	//Aktivera Utsignal Y1
	FB_MBReadCoils_Y1(
		sIPAddr:= sIpAddr, 
		nTCPPort:= INT_TO_UINT(nTCPPort), 
		nUnitID:= INT_TO_BYTE(nUnitID), 
		nQuantity:=1, 
		nMBAddr:= 0, 
		cbLength:= SIZEOF(bY1EnableRead), 
		pDestAddr:= ADR(bY1EnableRead), 
		bExecute:= bSekvensFlagga, 
		tTimeout:= T#3S, 
		bBusy=> , 
		bError=> , 
		nErrId=> , 
		cbRead=> );
				
		IF bY1Enable <> bY1EnableRead AND bSekvensFlagga THEN
			FB_MBWriteCoils_Y1.bExecute := TRUE;
		ELSE
			FB_MBWriteCoils_Y1.bExecute := FALSE;
		END_IF
		
	FB_MBWriteCoils_Y1(
		sIPAddr:= sIpAddr, 
		nTCPPort:= INT_TO_UINT(nTCPPort), 
		nUnitID:= INT_TO_BYTE(nUnitID), 
		nQuantity:= 1, 
		nMBAddr:= 0, 
		cbLength:= SIZEOF(bY1Enable), 
		pSrcAddr:= ADR(bY1Enable), 
		bExecute:= , 
		tTimeout:= , 
		bBusy=> , 
		bError=> , 
		nErrId=> );	
		
	//Aktivera Utsignal Y2
	FB_MBReadCoils_Y2(
		sIPAddr:= sIpAddr, 
		nTCPPort:= INT_TO_UINT(nTCPPort), 
		nUnitID:= INT_TO_BYTE(nUnitID), 
		nQuantity:=1, 
		nMBAddr:= 1, 
		cbLength:= SIZEOF(bY2EnableRead), 
		pDestAddr:= ADR(bY2EnableRead), 
		bExecute:= bSekvensFlagga, 
		tTimeout:= T#3S, 
		bBusy=> , 
		bError=> , 
		nErrId=> , 
		cbRead=> );
				
		IF bY2Enable <> bY2EnableRead AND bSekvensFlagga THEN
			FB_MBWriteCoils_Y2.bExecute := TRUE;
		ELSE
			FB_MBWriteCoils_Y2.bExecute := FALSE;
		END_IF
		
	FB_MBWriteCoils_Y2(
		sIPAddr:= sIpAddr, 
		nTCPPort:= INT_TO_UINT(nTCPPort), 
		nUnitID:= INT_TO_BYTE(nUnitID), 
		nQuantity:= 1, 
		nMBAddr:= 1, 
		cbLength:= SIZEOF(bY2Enable), 
		pSrcAddr:= ADR(bY2Enable), 
		bExecute:= , 
		tTimeout:= , 
		bBusy=> , 
		bError=> , 
		nErrId=> );		
		
	//Aktivera Utsignal Y3
	FB_MBReadCoils_Y3(
		sIPAddr:= sIpAddr, 
		nTCPPort:= INT_TO_UINT(nTCPPort), 
		nUnitID:= INT_TO_BYTE(nUnitID), 
		nQuantity:=1, 
		nMBAddr:= 2, 
		cbLength:= SIZEOF(bY3EnableRead), 
		pDestAddr:= ADR(bY3EnableRead), 
		bExecute:= bSekvensFlagga, 
		tTimeout:= T#3S, 
		bBusy=> , 
		bError=> , 
		nErrId=> , 
		cbRead=> );
				
		IF bY3Enable <> bY3EnableRead AND bSekvensFlagga THEN
			FB_MBWriteCoils_Y3.bExecute := TRUE;
		ELSE
			FB_MBWriteCoils_Y3.bExecute := FALSE;
		END_IF
		
	FB_MBWriteCoils_Y3(
		sIPAddr:= sIpAddr, 
		nTCPPort:= INT_TO_UINT(nTCPPort), 
		nUnitID:= INT_TO_BYTE(nUnitID), 
		nQuantity:= 1, 
		nMBAddr:= 2, 
		cbLength:= SIZEOF(bY3Enable), 
		pSrcAddr:= ADR(bY3Enable), 
		bExecute:= , 
		tTimeout:= , 
		bBusy=> , 
		bError=> , 
		nErrId=> );		
		
	//Aktivera Utsignal Y4
	FB_MBReadCoils_Y4(
		sIPAddr:= sIpAddr, 
		nTCPPort:= INT_TO_UINT(nTCPPort), 
		nUnitID:= INT_TO_BYTE(nUnitID), 
		nQuantity:=1, 
		nMBAddr:= 3, 
		cbLength:= SIZEOF(bY4EnableRead), 
		pDestAddr:= ADR(bY4EnableRead), 
		bExecute:= bSekvensFlagga, 
		tTimeout:= T#3S, 
		bBusy=> , 
		bError=> , 
		nErrId=> , 
		cbRead=> );
				
		IF bY4Enable <> bY4EnableRead AND bSekvensFlagga THEN
			FB_MBWriteCoils_Y4.bExecute := TRUE;
		ELSE
			FB_MBWriteCoils_Y4.bExecute := FALSE;
		END_IF
		
	FB_MBWriteCoils_Y4(
		sIPAddr:= sIpAddr, 
		nTCPPort:= INT_TO_UINT(nTCPPort), 
		nUnitID:= INT_TO_BYTE(nUnitID), 
		nQuantity:= 1, 
		nMBAddr:= 3, 
		cbLength:= SIZEOF(bY4Enable), 
		pSrcAddr:= ADR(bY4Enable), 
		bExecute:= , 
		tTimeout:= , 
		bBusy=> , 
		bError=> , 
		nErrId=> );		

//Holding register

//Börvärde Y1
wTemp := OaksLibrary.fRealToWord(rReal:= rY1Setpoint, uiFaktor:= 10);
//rtemp := rY1Setpoint * 10;
//iTemp := LIMIT(0,REAL_TO_UINT(rtemp),1000);
		
//Skriv börvärde
fbReadWriteHoldingReg_Y1(
	sIPAddr:= sIpAddr, 
	nTCPPort:= INT_TO_UINT(nTCPPort), 
	nUnitID:= INT_TO_BYTE(nUnitID), 
	mBusAdr:= 0, 
	bEnable:= bSekvensFlagga AND bY1Enable, 
	iWrite:= wTemp, 
	iRead=> , 
	bError=> );

//Börvärde Y2
wTemp := OaksLibrary.fRealToWord(rReal:= rY2Setpoint, uiFaktor:= 10);
//rtemp := rY2Setpoint * 10;
//iTemp := LIMIT(0,REAL_TO_UINT(rtemp),1000);
		
//Skriv börvärde Setpoint
fbReadWriteHoldingReg_Y2(
	sIPAddr:= sIpAddr, 
	nTCPPort:= INT_TO_UINT(nTCPPort), 
	nUnitID:= INT_TO_BYTE(nUnitID), 
	mBusAdr:= 1, 
	bEnable:= bSekvensFlagga AND bY2Enable, 
	iWrite:= wTemp, 
	iRead=> , 
	bError=> );	

//Börvärde Y3
wTemp := OaksLibrary.fRealToWord(rReal:= rY3Setpoint, uiFaktor:= 10);	
//rtemp := rY3Setpoint * 10;
//iTemp := LIMIT(0,REAL_TO_UINT(rtemp),1000);
		
//Skriv börvärde Setpoint
fbReadWriteHoldingReg_Y3(
	sIPAddr:= sIpAddr, 
	nTCPPort:= INT_TO_UINT(nTCPPort), 
	nUnitID:= INT_TO_BYTE(nUnitID), 
	mBusAdr:= 2, 
	bEnable:= bSekvensFlagga AND bY3Enable, 
	iWrite:= wTemp, 
	iRead=> , 
	bError=> );	
	
//Börvärde Y4
wTemp := OaksLibrary.fRealToWord(rReal:= rY4Setpoint, uiFaktor:= 10);	
//rtemp := rY4Setpoint * 10;
//iTemp := LIMIT(0,REAL_TO_UINT(rtemp),1000);
		
//Skriv börvärde Setpoint
fbReadWriteHoldingReg_Y4(
	sIPAddr:= sIpAddr, 
	nTCPPort:= INT_TO_UINT(nTCPPort), 
	nUnitID:= INT_TO_BYTE(nUnitID), 
	mBusAdr:= 3, 
	bEnable:= bSekvensFlagga AND bY4Enable, 
	iWrite:= wTemp, 
	iRead=> , 
	bError=> );	
	
//Communication error
	fbKommTof(IN:=FB_MBReadRegs_InputRegs1.bError OR FB_MBReadCoils_Y1.bError OR FB_MBReadCoils_Y2.bError OR FB_MBReadCoils_Y3.bError OR FB_MBReadCoils_Y4.bError OR fbReadWriteHoldingReg_Y1.bError OR fbReadWriteHoldingReg_Y2.bError OR fbReadWriteHoldingReg_Y3.bError OR fbReadWriteHoldingReg_Y4.bError, PT:=T#20S , Q=> , ET=> );
	
	fbAlarm_1(bInput:= fbKommTof.Q, tAlarmDelay:= T#20M, bAutoReset:= TRUE, bAlarmOutput=> FAULT);
		
//Write busy	
	oaksgvl.aBModbusBusyFlagga[iModbusLoop,nUnitID] := FB_MBReadRegs_InputRegs1.bBusy OR FB_MBReadCoils_Y1.bBusy OR FB_MBReadCoils_Y2.bBusy OR FB_MBReadCoils_Y3.bBusy OR FB_MBReadCoils_Y4.bBusy OR fbReadWriteHoldingReg_Y1.bBusy OR fbReadWriteHoldingReg_Y2.bBusy OR fbReadWriteHoldingReg_Y3.bBusy OR fbReadWriteHoldingReg_Y4.bBusy;

END_FUNCTION_BLOCK

// oaksModbusLibrary/Produal/Regulatorer/fbProdualHdhmCo2PirOverride
FUNCTION_BLOCK fbProdualHdhmCo2PirOverride EXTENDS fbProdualHdhmCo2Override
VAR_INPUT 
END_VAR
VAR_OUTPUT
	V AT %M*: BOOL; //Närvaroindikering (fördröjt till och frånslag)~wp:[trendoptions]i:300
	PV4 AT %M*: BOOL; //Närvarogivare (Rå-värde)~wp:[trendoptions]i:300	
END_VAR
VAR
	fbReadPir : FB_MBReadInputs;
	
	fbWriteStartDelay : fbReadWriteHoldingRegReal;
	fbWriteStopDelay : fbReadWriteHoldingRegReal;
	bReadPir : BYTE; // 10002 PIR sensor state (immediate) - 10003 PIR sensor state (control)
END_VAR

VAR_INPUT PERSISTENT
	SP7 AT %M*: REAL; //Fördröjning aktivering närvaroindikering (0-1-2)~wp:[format]0
	SP8 AT %M*: REAL; //Fördröjning inaktivering närvaroindikering (0-1-2-3-4-5)~wp:[format]0
END_VAR

SUPER^();

	//Read Status
	fbReadPir(
	sIPAddr:= sIpAddr, 
	nTCPPort:= INT_TO_UINT(nTCPPort), 
	nUnitID:= INT_TO_BYTE(nUnitID), 
	nQuantity:= 2, 
	nMBAddr:= 1, 
	cbLength:= SIZEOF(bReadPir), 
	pDestAddr:= ADR(bReadPir), 
	bExecute:= bSekvensFlagga, 
	tTimeout:=T#20S , 
	bBusy=> , 
	bError=> , 
	nErrId=> , 
	cbRead=> );
	
	PV4 :=  bReadPir.0;
	V := bReadPir.1;

	//Start-/Stoppfördröjning
	
	fbWriteStartDelay(
	sIPAddr:= sIpAddr, 
	nTCPPort:= INT_TO_UINT(nTCPPort), 
	nUnitID:= INT_TO_BYTE(nUnitID), 
	mBusAdr:=34 , 
	bEnable:=bSekvensFlagga , 
	tTimeout:= T#3S, 
	rReal:= SP7, 
	uiFaktor:= 1, 
	bError=> , 
	bBusy=> , 
	bSuccess=> );
		
	fbWriteStopDelay(
	sIPAddr:= sIpAddr, 
	nTCPPort:= INT_TO_UINT(nTCPPort), 
	nUnitID:= INT_TO_BYTE(nUnitID), 
	mBusAdr:=35 , 
	bEnable:=bSekvensFlagga , 
	tTimeout:= T#3S, 
	rReal:= SP8, 
	uiFaktor:= 1, 
	bError=> , 
	bBusy=> , 
	bSuccess=> );

END_FUNCTION_BLOCK

// oaksModbusLibrary/Regin/Givare/fbCthrc
FUNCTION_BLOCK fbCthrc
VAR_INPUT
	sIPAddr : STRING := ''; 
	nTCPPort : UINT;
	nUnitID : UINT;
	iModbusLoop : INT :=1; //Modbusslinga
	tKommfelsLarm : TIME := T#20M;
END_VAR
VAR_OUTPUT
	PV AT %M* : REAL;//Rumstemperatur~wp:[unit]°C[format]0.0[trendoptions]i:300
	PV1 AT %M* : REAL;//Koldioxidhalt~wp:[unit]ppm[format]0[trendoptions]i:300
	PV2 AT %M* : REAL;//Fukthalt~wp:[unit]rH%[format]0[trendoptions]i:300
	PV8 AT %M* : STRING;//Modbus konfiguering~wp:
	FAULT AT %M* : BOOL;//Kommunikationsfel~wp:
END_VAR
VAR
	sIP: STRING(255);
	sPort: STRING(255);
	sModbusID: STRING(255);
	sModbusLoop: STRING(255);
	sTemp : STRING(255);

	rTemp : REAL;
	fbKommTof : tof; 
	fbKommTon : ton;
	fbTempCo2Humidity: FB_MBReadRegs;
	wTempCo2Humidity : ARRAY[0..2] OF WORD; 
	bSekvensFlagga : BOOL;
END_VAR

//Modbus konfiguering
	sIP := CONCAT (SIPAddr, '');
	sPort := CONCAT ('<br>Port: ', UINT_TO_STRING(nTCPPort)); 								
	sModbusID := CONCAT('<br>ID: ', UINT_TO_STRING(nUnitID));
	sModbusLoop := CONCAT('<br>Loop: ', INT_TO_STRING(iModbusLoop));	

	sTemp := sIP;
	sTemp := CONCAT(sTemp, sPort);
	sTemp := CONCAT(sTemp, sModbusID);
	sTemp := CONCAT(sTemp, sModbusLoop);
	
	PV8 := sTemp;

//Sekvens	
	bSekvensFlagga := oaksGVL.aBModbusSekvens[iModbusLoop] = UINT_TO_INT(nUnitID);	
	
fbTempCo2Humidity(
	sIPAddr:= sIpAddr, 
	nTCPPort:= INT_TO_UINT(nTCPPort), 
	nUnitID:= INT_TO_BYTE(nUnitID), 
	nQuantity:=3 , 
	nMBAddr:=3999 , 
	cbLength:= SIZEOF(wTempCo2Humidity), 
	pDestAddr:= ADR(wTempCo2Humidity), 
	bExecute:= bSekvensFlagga, 
	tTimeout:= T#4.5S, 
	bBusy=> , 
	bError=> , 
	nErrId=> , 
	cbRead=> );
	
	fbKommTof(IN:=fbTempCo2Humidity.bError , PT:=T#20S , Q=> , ET=> );
	fbKommTon(IN:=fbKommTof.Q , PT:=tKommfelsLarm , Q=> , ET=> );
	FAULT :=fbKommTon.Q;
	
	rTemp := wTempCo2Humidity[0];
	PV2 := rTemp / 10 ; 
	rTemp := wTempCo2Humidity[1];
	PV := rTemp / 10; 
	PV1 := wTempCo2Humidity[2];

	//Write busy	
	oaksgvl.aBModbusBusyFlagga[iModbusLoop,nUnitID] := fbTempCo2Humidity.bBusy;

END_FUNCTION_BLOCK

// oaksModbusLibrary/Regin/Givare/fbCtrc
FUNCTION_BLOCK fbCtrc
VAR_INPUT
	sIPAddr : STRING := ''; 
	nTCPPort : UINT;
	nUnitID : UINT;
	iModbusLoop : INT :=1; //Modbusslinga
	tKommfelsLarm : TIME := T#20M;
END_VAR
VAR_OUTPUT
	PV AT %M* : REAL;//Rumstemperatur~wp:[unit]°C[format]0.0[trendoptions]i:300
	PV1 AT %M* : REAL;//Koldioxidhalt~wp:[unit]ppm[trendoptions]i:300
	PV8 AT %M* : STRING;//Modbus konfiguering~wp:
	FAULT AT %M* : BOOL;//Kommunikationsfel~wp:


END_VAR
VAR
	sIP: STRING(255);
	sPort: STRING(255);
	sModbusID: STRING(255);
	sModbusLoop: STRING(255);
	sTemp : STRING(255);

	rTemp : REAL;
	fbKommTof : tof; 
	fbKommTon : ton;
	fbTempCo2Humidity: FB_MBReadRegs;
	wTempCo2Humidity : ARRAY[0..1] OF	WORD; 
	bSekvensFlagga : BOOL;
END_VAR

//Modbus konfiguering
	sIP := CONCAT (SIPAddr, '');
	sPort := CONCAT ('<br>Port: ', UINT_TO_STRING(nTCPPort)); 								
	sModbusID := CONCAT('<br>ID: ', UINT_TO_STRING(nUnitID));
	sModbusLoop := CONCAT('<br>Loop: ', INT_TO_STRING(iModbusLoop));	

	sTemp := sIP;
	sTemp := CONCAT(sTemp, sPort);
	sTemp := CONCAT(sTemp, sModbusID);
	sTemp := CONCAT(sTemp, sModbusLoop);
	
	PV8 := sTemp;

//Sekvens	
	bSekvensFlagga := oaksGVL.aBModbusSekvens[iModbusLoop] = UINT_TO_INT(nUnitID);	
	
fbTempCo2Humidity(
	sIPAddr:= sIpAddr, 
	nTCPPort:= INT_TO_UINT(nTCPPort), 
	nUnitID:= INT_TO_BYTE(nUnitID), 
	nQuantity:=2 , 
	nMBAddr:=4000 , 
	cbLength:= SIZEOF(wTempCo2Humidity), 
	pDestAddr:= ADR(wTempCo2Humidity), 
	bExecute:= bSekvensFlagga, 
	tTimeout:= T#3S, 
	bBusy=> , 
	bError=> , 
	nErrId=> , 
	cbRead=> );
	
	fbKommTof(IN:=fbTempCo2Humidity.bError , PT:=T#20S , Q=> , ET=> );
	fbKommTon(IN:=fbKommTof.Q , PT:=tKommfelsLarm , Q=> , ET=> );
	FAULT :=fbKommTon.Q;
	
	
	rTemp := wTempCo2Humidity[0];
	PV := rTemp / 10; 
	PV1 := wTempCo2Humidity[1];

	//Write busy	
	oaksgvl.aBModbusBusyFlagga[iModbusLoop,nUnitID] := fbTempCo2Humidity.bBusy;

END_FUNCTION_BLOCK

// oaksModbusLibrary/Regin/Regio midi/fbReginRCC
//OAKS AB
//2020-04-28
//Funktionsblock för modbus-TCP, Regin RCC-C3DOCS rumsreglator med kyla/värme/spjäll. Inbyggda larm för hög/låg rumstemperatur och hög CO2-halt.
FUNCTION_BLOCK fbReginRCC
VAR_INPUT
	sIPAddr : STRING := ''; 
	nTCPPort : UINT := 502;
	nUnitID : UINT :=1;
	iModbusLoop : INT :=1; //Modbusslinga
	bInvertVav : BOOL; // Invertering av VAV_OP används vid ändrad gångriktning på spjäll
	SP1 AT %M* : REAL;//Börvärde värme rumstemperatur~wp:[unit]°C[format]0.0
	SP2 AT %M* : REAL;//Börvärde kyla rumstemperatur~wp:[unit]°C[format]0.0
END_VAR

VAR_INPUT PERSISTENT
	AHL AT %M* : REAL := 23;//Larmgräns hög rumstemperatur~wp:[unit]°C[format]0.0
	ALL AT %M* : REAL := 18;//Larmgräns låg rumstemperatur~wp:[unit]°C[format]0.0
	AD AT %M* : REAL := 30;//Larmfördröjning låg/hög rumstemperatur~wp:[unit]min[format]0
	tTimeout : TIME := T#20M; 
END_VAR

VAR_OUTPUT
	PV AT %M* : REAL;//Rumstemperatur~wp:[unit]°C[format]0.0[trendoptions]i:300
	CSP AT %M* : REAL;//Uträknat börvärde rumstemperatur~wp:[unit]°C[format]0.0[trendoptions]i:300
	HEATING_OP AT %M* : REAL;//Utsignal värme~wp:[unit]%[format]0[trendoptions]i:300
	COOLING_OP AT %M* : REAL;//Utsignal kyla~wp:[unit]%[format]0[trendoptions]i:300
	VAV_OP AT %M* : REAL;//Utsignal spjällställdon~wp:[unit]%[format]0[trendoptions]i:300
			
	bRegioPresence AT %M* : BOOL;//Närvaroindikering	
	PV8 AT %M* : STRING;//Modbus konfiguering~wp:	
	FAULT AT %M* : BOOL;//Kommunikationsfel~wp:
	
	//Alarms
	HAL AT %M* : BOOL;//Hög rumstemperatur~wp:
	LAL AT %M* : BOOL;//Låg rumstemperatur~wp:
	
END_VAR

VAR
	//General
	offset : INT;
	rTemp : REAL;
	iTemp : INT;
	wTemp : WORD;
	bSekvensFlagga : BOOL;
	
	wRegioPresence : WORD;
				
	//Read input registers
	FB_MBReadInputRegs_wArrInput1: FB_MBReadInputRegs;
	wArrInputRegs1 : ARRAY [11..32] OF WORD; //Input register function 4

	FB_SETPOINT_INT_MODBUS_Heat : FB_SETPOINT_INT_MODBUS;
	//Skrivning heat setpoint 
	fbWriteHoldingDoubleControlledHeat: fbDoubleControlledModbusHolding;

	
	
	//Skrivning heat setpoint
	fbWriteHoldingDoubleControlledCool: fbDoubleControlledModbusHolding;
	
	//Skrivning heat min. CO2
	fbWriteHoldingDoubleControlledMinCO2: fbDoubleControlledModbusHolding;
	
	//Skrivning heat max. CO2
	fbWriteHoldingDoubleControlledMaxCO2: fbDoubleControlledModbusHolding;
	
	
	
	//Kommunikationsfel
	fbKommTof : tof; 
	fbKommTon : ton;

	bError: INT;
	
	//Alarms
	fbHighLimitAlarm_temp: fbHighLimitAlarm;
	fbLowLimitAlarm_temp: fbLowLimitAlarm;
	fbHighLimitAlarm_CO2: fbHighLimitAlarm;
	
	
	sIP: STRING(255);
	sPort: STRING(255);
	sModbusID: STRING(255);
	sModbusLoop: STRING(255);
	sTemp : STRING(255);
	
	FB_MBReadInputsPresence: FB_MBReadInputs;
END_VAR

//General
	offset := -1;
//Sekvens	
	bSekvensFlagga := oaksGVL.aBModbusSekvens[iModbusLoop] = UINT_TO_INT(nUnitID);

//Modbus konfiguering
	sIP := CONCAT (SIPAddr, '');
	sPort := CONCAT ('<br>Port: ', UINT_TO_STRING(nTCPPort)); 								
	sModbusID := CONCAT('<br>ID: ', UINT_TO_STRING(nUnitID));
	sModbusLoop := CONCAT('<br>Loop: ', INT_TO_STRING(iModbusLoop));

	sTemp := sIP;
	sTemp := CONCAT(sTemp, sPort);
	sTemp := CONCAT(sTemp, sModbusID);
	sTemp := CONCAT(sTemp, sModbusLoop);
		
	PV8 := sTemp;
	
///////////////		
//READ
///////////////			

	FB_MBReadInputsPresence(
	sIPAddr:= sIpAddr, 
	nTCPPort:= INT_TO_UINT(nTCPPort), 
	nUnitID:= INT_TO_BYTE(nUnitID), 
	nQuantity:= 1, 
	nMBAddr:= 30, 
	cbLength:= SIZEOF(wRegioPresence), 
	pDestAddr:= ADR(wRegioPresence), 
	bExecute:= bSekvensFlagga, 
	tTimeout:=T#10S , 
	bBusy=> , 
	bError=> , 
	nErrId=> , 
	cbRead=> );
	
	bRegioPresence := WORD_TO_BOOL(wRegioPresence);

		
//Read input registers function 4		

	//Read Array1
	FB_MBReadInputRegs_wArrInput1(
		sIPAddr:= sIpAddr, 
		nTCPPort:= INT_TO_UINT(nTCPPort), 
		nUnitID:= INT_TO_BYTE(nUnitID), 
		nQuantity:= 22, 
		nMBAddr:= 11 + offset, 
		cbLength:= SIZEOF(wArrInputRegs1), 
		pDestAddr:= ADR(wArrInputRegs1), 
		bExecute:= bSekvensFlagga, 
		tTimeout:= T#10S, 
		bBusy=> , 
		bError=> , 
		nErrId=> , 
		cbRead=> );
	
		//Values
		//wArrInputRegs1[1]; //1
		//wArrInputRegs1[2]; //2
		//wArrInputRegs1[3]; //3
		//wArrInputRegs1[4]; //4
		//wArrInputRegs1[5]; //5
		//wArrInputRegs1[6]; //6
		//wArrInputRegs1[7]); //7
		//wArrInputRegs1[8]; //8
		//wArrInputRegs1[9]; //9
		//wArrInputRegs1[10]; //10
		iTemp := WORD_TO_INT(wArrInputRegs1[11]); // Rumstemperatur
		PV := INT_TO_REAL(iTemp) /10;
		//wArrInputRegs1[12]; //12
		//wArrInputRegs1[13]; //12
		//wArrInputRegs1[14]; //14
		//wArrInputRegs1[15]; //15
		//wArrInputRegs1[16]; //16
		//wArrInputRegs1[17]; //17
		//wArrInputRegs1[18]; //18
		//wArrInputRegs1[19]); //19
		iTemp := WORD_TO_INT(wArrInputRegs1[20]); // Uträknat börvärde rumstemperatur
		
		CSP := INT_TO_REAL(iTemp) /10;
		
		//wArrInputRegs1[21]; //21
		
		iTemp := WORD_TO_INT(wArrInputRegs1[22]); //Utsignal värme
		HEATING_OP := INT_TO_REAL(iTemp);
		
		iTemp := WORD_TO_INT(wArrInputRegs1[23]); //Utsignal kyla		
		COOLING_OP := INT_TO_REAL(iTemp);

		//wArrInputRegs1[24]; //24
		//wArrInputRegs1[25]; //25
		
		iTemp := WORD_TO_INT(wArrInputRegs1[26]); //Utsignal spjällställdon
		IF NOT bInvertVav THEN 
			VAV_OP := INT_TO_REAL(iTemp);
		ELSE
			VAV_OP := INT_TO_REAL(100-iTemp);
		END_IF
		
		//wArrInputRegs1[27]; //27
		//wArrInputRegs1[28]; //28
		//wArrInputRegs1[29]; //29
		//wArrInputRegs1[30]; //30
		//wArrInputRegs1[31]; //31
		

		
		
//Read Holding registers function 3		
	

	
//Write Holding registers
	
	//Heat setpoint
	
	fbWriteHoldingDoubleControlledHeat(
	sIPAddr:=sIPAddr , 
	nTCPPort:=nTCPPort , 
	nUnitID:= UINT_TO_BYTE(nUnitID), 
	nMBAddr:=68+offset , 
	bExecute:=bSekvensFlagga , 
	rScale:=10 , 
	rWrite:= SP1, 
	bBusy=> );
	
	//Cool setpoint
	fbWriteHoldingDoubleControlledCool(
	sIPAddr:= sIPAddr, 
	nTCPPort:= nTCPPort, 
	nUnitID:= UINT_TO_BYTE(nUnitID) , 
	nMBAddr:= 69+offset, 
	bExecute:=bSekvensFlagga , 
	rScale:= 10, 
	rWrite:=SP2 , 
	bBusy=> );
		
		

	
//Alarms

	fbHighLimitAlarm_temp(
		//bInput:= , 
		tAlarmDelay:= REAL_TO_TIME(AD * 60000), 
		bAutoReset:= TRUE, 
		bAlarmOutput=> HAL, 
		bEnable:= TRUE AND NOT FAULT, 
		rProcessValue:= PV, 
		rHighLimit:= AHL);
		
	fbLowLimitAlarm_temp(
		//bInput:= , 
		tAlarmDelay:= REAL_TO_TIME(AD * 60000), 
		bAutoReset:= TRUE, 
		bAlarmOutput=> LAL, 
		bEnable:= TRUE AND NOT FAULT, 
		rProcessValue:= PV, 
		rLowLimit:= ALL);
	

	
//Communication error
	fbKommTof(IN:= FB_MBReadInputRegs_wArrInput1.bError OR
		fbWriteHoldingDoubleControlledHeat.bError OR
		fbWriteHoldingDoubleControlledCool.bError OR
		fbWriteHoldingDoubleControlledMinCO2.bError OR
		fbWriteHoldingDoubleControlledMaxCO2.bError,
		PT:=T#20S , Q=> , ET=> );
		fbKommTon(IN:=fbKommTof.Q , PT:=tTimeout , Q=> , ET=> );
		FAULT :=fbKommTon.Q;

//Write busy	
	oaksgvl.aBModbusBusyFlagga[iModbusLoop,nUnitID] := FB_MBReadInputRegs_wArrInput1.bBusy OR
		fbWriteHoldingDoubleControlledHeat.bBusy OR
		fbWriteHoldingDoubleControlledCool.bBusy OR
		fbWriteHoldingDoubleControlledMinCO2.bBusy OR
		fbWriteHoldingDoubleControlledMaxCO2.bBusy;

END_FUNCTION_BLOCK

// oaksModbusLibrary/Regin/Regio midi/fbReginRCC_CO2
FUNCTION_BLOCK fbReginRCC_CO2 EXTENDS fbReginRCC
VAR_INPUT
	SP3 AT %M* : REAL;//Min. CO2-halt~wp:[unit]ppm[format]0
	SP4 AT %M* : REAL;//Max. CO2-halt~wp:[unit]ppm[format]0
END_VAR
VAR_OUTPUT
	PV1 AT %M* : REAL;//Koldioxid~wp:[unit]ppm[format]0[trendoptions]i:300
	AL AT %M* : BOOL;//Hög CO2-halt~wp:
END_VAR
VAR_INPUT PERSISTENT 
	AHHL AT %M* : REAL := 1000;//Larmgräns hög CO2-halt~wp:[unit]ppm[format]0
	HAD AT %M* : REAL := 30;//Larmfördröjning CO2-halt~wp:[unit]min[format]0
END_VAR

SUPER^();

	iTemp := WORD_TO_INT(wArrInputRegs1[32]); //Koldioxidhalt
	PV1 := INT_TO_REAL(iTemp);

	//Min C02
	fbWriteHoldingDoubleControlledMinCO2(
	sIPAddr:= sIPAddr, 
	nTCPPort:= nTCPPort, 
	nUnitID:= UINT_TO_BYTE(nUnitID) , 
	nMBAddr:= 147+offset, 
	bExecute:=bSekvensFlagga , 
	rScale:=1 , 
	rWrite:=SP3 , 
	bBusy=> );


	//Max setpoint
	
	fbWriteHoldingDoubleControlledMaxCO2(
	sIPAddr:= sIPAddr, 
	nTCPPort:= nTCPPort, 
	nUnitID:= UINT_TO_BYTE(nUnitID) , 
	nMBAddr:=148+offset , 
	bExecute:= bSekvensFlagga, 
	rScale:= 1, 
	rWrite:= SP4, 
	bBusy=> );

	fbHighLimitAlarm_CO2(
		//bInput:= , 
		tAlarmDelay:= REAL_TO_TIME(HAD * 60000), 
		bAutoReset:= TRUE, 
		bAlarmOutput=> AL, 
		bEnable:= TRUE AND NOT FAULT, 
		rProcessValue:= PV1, 
		rHighLimit:= AHHL);

END_FUNCTION_BLOCK

// oaksModbusLibrary/Regin/Regio midi/fbReginRCC_Handst_Spjall
//OAKS AB
//2020-04-28
//Funktionsblock för modbus-TCP, Regin RCC-C3DOCS rumsreglator med kyla/värme/spjäll. Funktion för lolak regulator i plc och handställning av utgångar.
FUNCTION_BLOCK fbReginRCC_Handst_Spjall
VAR_INPUT
	bForcera : BOOL; // Forcera 100% öppet
	sIPAddr : STRING := ''; 
	nTCPPort : UINT := 502;
	nUnitID : UINT :=1;
	iModbusLoop : INT :=1; //Modbusslinga
	bInvertVav : BOOL; // Invertering av VAV_OP används vid ändrad gångriktning på spjäll
END_VAR

VAR_INPUT PERSISTENT
	SP AT %M* : REAL := 22;//Börvärde rumstemperatur~wp:[unit]°C[format]0.0
	P  AT %M* : REAL := 1;  //Förstärkning regulator temperatur~wp:[format]0.00
	I  AT %M* : UDINT := 30; //I-tid regulator temperatur ~wp:
	AHL AT %M* : REAL := 25;//Larmgräns hög rumstemperatur~wp:[unit]°C[format]0.0
	ALL AT %M* : REAL := 15;//Larmgräns låg rumstemperatur~wp:[unit]°C[format]0.0
	AD AT %M* : REAL := 30;//Larmfördröjning låg/hög larm~wp:[unit]min[format]0
	tTimeout : TIME := T#20M;
END_VAR

VAR_OUTPUT
	PV AT %M* : REAL;//Rumstemperatur~wp:[unit]°C[format]0.0[trendoptions]i:300
	VAV_OP AT %M* : REAL;//Utsignal spjällställdon~wp:[unit]%[format]0[trendoptions]i:300
	PV8 AT %M* : STRING;//Modbus konfiguering~wp:	
	FAULT AT %M* : BOOL;//Kommunikationsfel~wp:
	
	//Alarms
	HAL AT %M* : BOOL;//Hög rumstemperatur~wp:
	LAL AT %M* : BOOL;//Låg rumstemperatur~wp:
	
END_VAR

VAR
	//General
	offset : INT;
	rTemp : REAL;
	iTemp : INT;
	wTemp : WORD;
	bSekvensFlagga : BOOL;
	
	wRegioPresence : WORD;
				
	//Read input registers
	FB_MBReadInputRegs_wArrInput1: FB_MBReadInputRegs;
	wArrInputRegs1 : ARRAY [11..32] OF WORD; //Input register function 4

	FB_SETPOINT_INT_MODBUS_Heat : FB_SETPOINT_INT_MODBUS;
	
	
	//Kommunikationsfel
	fbKommTof : tof; 
	fbKommTon : ton;

	bError: INT;
	
	//Alarms
	fbHighLimitAlarm_temp: fbHighLimitAlarm;
	fbLowLimitAlarm_temp: fbLowLimitAlarm;
	
	
	sIP: STRING(255);
	sPort: STRING(255);
	sModbusID: STRING(255);
	sModbusLoop: STRING(255);
	sTemp : STRING(255);
	
	FB_MBReadInputsPresence: FB_MBReadInputs;
	
	fbReadWriteHoldingRegHandstallning  : fbReadWriteHoldingReg;
	
	fbReadWriteHoldingRegHandstallningUtsignal  : fbReadWriteHoldingReg;
	
	fbControllerTemperature : fbController;
	
	uiInternvariabelCo2 : UINT; // Internvariabel skrivs till från extendat block med co2-regulator (fbReginRCC_Handst_Spjall_Co2)
END_VAR

//General
	offset := -1;
//Sekvens	
	bSekvensFlagga := oaksGVL.aBModbusSekvens[iModbusLoop] = UINT_TO_INT(nUnitID);

//Modbus konfiguering
	sIP := CONCAT (SIPAddr, '');
	sPort := CONCAT ('<br>Port: ', UINT_TO_STRING(nTCPPort)); 								
	sModbusID := CONCAT('<br>ID: ', UINT_TO_STRING(nUnitID));
	sModbusLoop := CONCAT('<br>Loop: ', INT_TO_STRING(iModbusLoop));

	sTemp := sIP;
	sTemp := CONCAT(sTemp, sPort);
	sTemp := CONCAT(sTemp, sModbusID);
	sTemp := CONCAT(sTemp, sModbusLoop);
		
	PV8 := sTemp;
		
//Read input registers function 4		

	fbControllerTemperature(
	bEnable:=TRUE , 
	rProcessValue:= PV, 
	rSetpoint:= SP, 
	bActn:= TRUE, 
	rKp:= P, 
	rKi:= I, 
	rDz:= , 
	rMin:= 0, 
	rMax:=100 , 
	rOutput=> );

// Handställning spjäll Handställning Spjäll  Handställning (2=AUT) // 11
	fbReadWriteHoldingRegHandstallning(
	sIPAddr:= sIpAddr, 
	nTCPPort:= INT_TO_UINT(nTCPPort), 
	nUnitID:= INT_TO_BYTE(nUnitID), 
	mBusAdr:= 11, 
	bEnable:=bSekvensFlagga, 
	iWrite:= 1, 
	iRead=> , 
	bError=> , 
	bBusy=> );

// Manuell Utsignal Spjäll % holding 92
	IF NOT bForcera THEN
		fbReadWriteHoldingRegHandstallning.iWrite := MAX(REAL_TO_UINT(fbControllerTemperature.rOutput),uiInternvariabelCo2);
	ELSE
		fbReadWriteHoldingRegHandstallning.iWrite := 100;
	END_IF

	fbReadWriteHoldingRegHandstallning(
	sIPAddr:= sIpAddr, 
	nTCPPort:= INT_TO_UINT(nTCPPort), 
	nUnitID:= INT_TO_BYTE(nUnitID), 
	mBusAdr:= 92, 
	bEnable:=bSekvensFlagga,  
	iRead=> , 
	bError=> , 
	bBusy=> );

	//Read Array1
	FB_MBReadInputRegs_wArrInput1(
		sIPAddr:= sIpAddr, 
		nTCPPort:= INT_TO_UINT(nTCPPort), 
		nUnitID:= INT_TO_BYTE(nUnitID), 
		nQuantity:= 22, 
		nMBAddr:= 11 + offset, 
		cbLength:= SIZEOF(wArrInputRegs1), 
		pDestAddr:= ADR(wArrInputRegs1), 
		bExecute:= bSekvensFlagga, 
		tTimeout:= T#3S, 
		bBusy=> , 
		bError=> , 
		nErrId=> , 
		cbRead=> );
	
		iTemp := WORD_TO_INT(wArrInputRegs1[11]); // Rumstemperatur
		PV := INT_TO_REAL(iTemp) /10;

		
		iTemp := WORD_TO_INT(wArrInputRegs1[26]); //Utsignal spjällställdon
		IF NOT bInvertVav THEN 
			VAV_OP := INT_TO_REAL(iTemp);
		ELSE
			VAV_OP := INT_TO_REAL(100-iTemp);
		END_IF
		
		

//Alarms

	fbHighLimitAlarm_temp(
		//bInput:= , 
		tAlarmDelay:= REAL_TO_TIME(AD * 60000), 
		bAutoReset:= TRUE, 
		bAlarmOutput=> HAL, 
		bEnable:= TRUE AND NOT FAULT, 
		rProcessValue:= PV, 
		rHighLimit:= AHL);
		
	fbLowLimitAlarm_temp(
		//bInput:= , 
		tAlarmDelay:= REAL_TO_TIME(AD * 60000), 
		bAutoReset:= TRUE, 
		bAlarmOutput=> LAL, 
		bEnable:= TRUE AND NOT FAULT, 
		rProcessValue:= PV, 
		rLowLimit:= ALL);
	

	
//Communication error
	fbKommTof(IN:= FB_MBReadInputRegs_wArrInput1.bError, PT:=T#20S , Q=> , ET=> );
	fbKommTon(IN:=fbKommTof.Q , PT:=tTimeout , Q=> , ET=> );
	FAULT :=fbKommTon.Q;

//Write busy	
	oaksgvl.aBModbusBusyFlagga[iModbusLoop,nUnitID] := FB_MBReadInputRegs_wArrInput1.bBusy;

END_FUNCTION_BLOCK

// oaksModbusLibrary/Regin/Regio midi/fbReginRCC_Handst_Spjall_Co2
// Extendat block från fbReginRCC_Handst_Spjall med co2-reglering
FUNCTION_BLOCK fbReginRCC_Handst_Spjall_Co2 EXTENDS fbReginRCC_Handst_Spjall
VAR_INPUT
END_VAR
VAR_OUTPUT
	HHAL AT %M* : BOOL;//Hög co2-halt~wp:
	PV1 AT %M* : REAL;//Co2-halt~wp:[unit]ppm[format]0[trendoptions]i:300
END_VAR
VAR
	fbControllerCo2 : fbController;
	fbHighLimitAlarm_co2: fbHighLimitAlarm;
END_VAR
VAR_INPUT PERSISTENT
	SP1 AT %M* : REAL := 800;//Börvärde co2-halt~wp:[unit]ppm[format]0
	SP2  AT %M* : REAL := 1;  //Förstärkning regulator co2~wp:[format]0.00
	SP3  AT %M* : UDINT := 30; //I-tid regulator co2 ~wp:
	AHHL AT %M* : REAL := 1000;//Larmgräns hög co2-halt~wp:[unit]ppm[format]0
END_VAR

	SUPER^();
	iTemp := WORD_TO_INT(wArrInputRegs1[32]); //Koldioxidhalt
	PV1 := INT_TO_REAL(iTemp);

	fbControllerCo2(
	bEnable:=TRUE , 
	rProcessValue:= PV1, 
	rSetpoint:= SP1, 
	bActn:= TRUE, 
	rKp:= SP2, 
	rKi:= SP3, 
	rDz:= , 
	rMin:= 0, 
	rMax:=100 , 
	rOutput=> );
	
	uiInternvariabelCo2 := REAL_TO_UINT(fbControllerCo2.rOutput); 
	
		fbHighLimitAlarm_co2(
		//bInput:= , 
		tAlarmDelay:= REAL_TO_TIME(AD * 60000), 
		bAutoReset:= TRUE, 
		bAlarmOutput=> HHAL, 
		bEnable:= TRUE AND NOT FAULT, 
		rProcessValue:= PV1, 
		rHighLimit:= AHHL);

END_FUNCTION_BLOCK

// oaksModbusLibrary/Schneider/fbAltivarATV600
//Funktionsblock för kommunikation mot Altivar ATV600. Skriv larmreset, läsning av div. värden
//Robert H Oaks AB 
//22-03-22

//V 1.0	Testad

//OBS! Ej anpassad för Modbus-sekvens i oaks-standard, bör åtgärdas!!

FUNCTION_BLOCK fbAltivarATV600
VAR_INPUT
	sIPAddr 		: STRING; 			//Ip-adress till ModbusTCP-gateway
	nMBTCPPort		: UINT := 502;		//ModbusTCP-port
	nUnitID			: UINT := 1;		//Enhetsadress
	tInterval		: TIME := T#10S;	//Kommunikationsintervall
	tTimeout		: TIME := T#2S;		//Timeout
	CMD AT %M*		: BOOL;				//Larmreset ~wp:
	RST AT %M*		: BOOL;				//Reset drifttid ~wp:
END_VAR

VAR_OUTPUT
	AL		AT %M*		: BOOL;				//Larm (fel) frekv.omf~wp:[alarmoptions]p:2
	AL1		AT %M*		: BOOL;				//Larm (varning) frekv.omf~wp:[alarmoptions]p:3
	AL2		AT %M*		: BOOL;				//Frekv.omf lokalt stoppad~wp:[alarmoptions]p:3
	V1		AT %M*		: BOOL;				//Referens uppnådd~wp:[trendoptions]i:14400, t:1 
	V2		AT %M*		: BOOL;				//Strömbegränsning aktiv~wp:[trendoptions]i:14400, t:1
	V3		AT %M*		: BOOL;				//STO utlöst~wp:[trendoptions]i:14400, t:1
	PV		AT %M* 		: STRING := ''; 	//Driftläge~wp:[trendoptions]i:14400, t:1
	PV1		AT %M* 		: REAL; 			//Motorhastighet~wp:[unit]rpm[format]0[trendoptions]i:300
	PV2		AT %M* 		: REAL; 			//Motorfrekvens~wp:[unit]Hz[format]0.0[trendoptions]i:300
	PV3		AT %M* 		: REAL; 			//Motorström~wp:[unit]A[format]0.0[trendoptions]i:300
	PV4		AT %M* 		: REAL; 			//Motorspänning~wp:[unit]V[format]0[trendoptions]i:300
	PV5		AT %M* 		: REAL; 			//Effektförbrukning motor~wp:[unit]kW[format]0[trendoptions]i:300
	PV6		AT %M* 		: REAL; 			//Avgiven effekt motor~wp:[unit]kW[format]0[trendoptions]i:300
	PV7		AT %M* 		: REAL; 			//Effektbelastning motor~wp:[unit]%[format]0[trendoptions]i:300
	PV8		AT %M* 		: REAL; 			//Termisk belastning motor~wp:[unit]%[format]0[trendoptions]i:300
	PV9		AT %M* 		: REAL; 			//Termisk belastning frekv.omf~wp:[unit]%[format]0[trendoptions]i:300
	PV11	AT %M* 		: REAL; 			//Verkningsgrad motor~wp:[unit]%[format]0[trendoptions]i:300
	PV12	AT %M* 		: REAL; 			//Drifttid elektronik frekv.omf~wp:[unit]timmar[format]0[trendoptions]i:300
	PV13	AT %M* 		: REAL; 			//Antal motorstarter~wp:[unit]st[format]0[trendoptions]i:300
	PV14	AT %M* 		: UINT; 			//Aktuell felkod (se ERRD)~wp:[trendoptions]i:14400, t:1
	PV15	AT %M* 		: UINT; 			//Senaste felkod (se LFT)~wp:[trendoptions]i:14400, t:1
	PV16	AT %M* 		: UINT; 			//Felräknare~wp:[unit]st[format]0[trendoptions]i:300
	PV17	AT %M* 		: DINT; 			//Energiförbrukning ~wp:[unit]kWh[format]0[trendoptions]i:300
	
	AL8		AT %M*		: BOOL;				//Kommunikationsfel frekv.omf~wp:[alarmoptions]p:3
END_VAR

VAR
	bRun			: BOOL;	
	fbRunTON		: TON;
	fbRunTRIG		: R_TRIG;
	
	bDidRead		: BOOL;

	fbR8501			: FB_MBReadRegs;
	fbW8501			: FB_MBWriteSingleReg;
	fbW3120			: FB_MBWriteSingleReg;
	
	fbR3201			: FB_MBReadRegs;
	fbR3206			: FB_MBReadRegs;
	fbR8604			: FB_MBReadRegs;
	fbR3202			: FB_MBReadRegs;
	fbR3204			: FB_MBReadRegs;
	fbR3208			: FB_MBReadRegs;
	fbR3211			: FB_MBReadRegs;
	fbR3209			: FB_MBReadRegs;
	fbR3240			: FB_MBReadRegs;
	fbR9630			: FB_MBReadRegs;
	fbR8606			: FB_MBReadRegs;
	fbR7121			: FB_MBReadRegs;
	fbR7393			: FB_MBReadRegs;
	fbR15322		: FB_MBReadRegs;
	fbR16050		: FB_MBReadRegs;
	fbR3293			: FB_MBReadRegs;
	fbR3260_61		: FB_MBReadRegs;
	fbR10627		: FB_MBReadRegs;
	fbR10628		: FB_MBReadRegs;
	fbR10629		: FB_MBReadRegs;
	fbR3292			: FB_MBReadRegs;
	fbR3276_77		: FB_MBReadRegs;
	
	wR8501			: WORD;
	wR3201			: WORD;
	wR3206			: WORD;
	wR8604			: WORD;
	wR3202			: WORD;
	wR3204			: WORD;
	wR3208			: WORD;
	wR3211			: WORD;
	wR3209			: WORD;
	wR3240			: WORD;
	wR9630			: WORD;
	wR8606			: WORD;
	wR7121			: WORD;
	wR7393			: WORD;
	wR15322			: WORD;
	wR16050			: WORD;
	wR3293			: WORD;
	wR3292			: WORD;
	wR10627			: WORD;
	wR10628			: WORD;
	wR10629			: WORD;
	
	uR3260_61		: WORD2_TO_UDINT;
	uR3276_77		: WORD2_TO_UDINT;	
	
	fbErrorTOF		: TOF;
	fbErrorTON		: TON;
END_VAR

fbRunTON(IN := NOT bRun, PT := tInterval);
fbRunTRIG(CLK := fbRunTON.Q, Q => bRun);


//Command register			Endast larmreset. Läs in ord, då larmreset sätts från Webport skrivs ord tillbaks lika läsning med bit för larmreset hög	
IF CMD AND bRun THEN
	
	IF NOT bDidRead THEN
		fbR8501(sIPAddr := sIPAddr, nTCPPort := nMBTCPPort, nUnitID := UINT_TO_BYTE(nUnitID), nQuantity := 1, bExecute := bRun, tTimeout := tTimeout,   
			nMBAddr 	:= 8501,
			cbLength	:= SIZEOF(wR8501),
			pDestAddr	:= ADR(wR8501));
			
		bDidRead := TRUE;
	ELSE
		fbR8501(bExecute := FALSE);	//Uppdatera status
		IF NOT (fbR8501.bBusy OR fbR8501.bError) THEN
		
			wR8501.7 := TRUE;
		
			fbW8501(sIPAddr := sIPAddr, nTCPPort := nMBTCPPort, nUnitID := UINT_TO_BYTE(nUnitID), tTimeout := tTimeout,
				bExecute 	:= bRun,   
				nMBAddr 	:= 8501,
				nValue		:= wR8501);
				
			bDidRead	:= FALSE;
			CMD 		:= FALSE;			
		END_IF
	END_IF;			
ELSE
	fbW8501(bExecute := FALSE);
	fbR8501(bExecute := FALSE);
END_IF;

//Time counter reset		Återställ alla räknare genom att sätta enum=64
IF RST AND bRun THEN
	fbW3120(sIPAddr := sIPAddr, nTCPPort := nMBTCPPort, nUnitID := UINT_TO_BYTE(nUnitID), tTimeout := tTimeout,
		bExecute 	:= bRun,   
		nMBAddr 	:= 3120,
		nValue		:= 64);
		
	RST := FALSE;
ELSE
	fbW3120(bExecute := FALSE);
END_IF

//CIA402 State register	
fbR3201(sIPAddr := sIPAddr, nTCPPort := nMBTCPPort, nUnitID := UINT_TO_BYTE(nUnitID), nQuantity := 1, bExecute := bRun, tTimeout := tTimeout,   
	nMBAddr 	:= 3201,
	cbLength	:= SIZEOF(wR3201),
	pDestAddr	:= ADR(wR3201));
	AL1		:= wR3201.7;
	V1		:= wR3201.10;
	AL2		:= wR3201.14;
	
//Internal State register	
fbR3206(sIPAddr := sIPAddr, nTCPPort := nMBTCPPort, nUnitID := UINT_TO_BYTE(nUnitID), nQuantity := 1, bExecute := bRun, tTimeout := tTimeout,   
	nMBAddr 	:= 3206,
	cbLength	:= SIZEOF(wR3206),
	pDestAddr	:= ADR(wR3206));
	V2		:= wR3206.11;
	
//Output velocity	
fbR8604(sIPAddr := sIPAddr, nTCPPort := nMBTCPPort, nUnitID := UINT_TO_BYTE(nUnitID), nQuantity := 1, bExecute := bRun, tTimeout := tTimeout,   
	nMBAddr 	:= 8604,
	cbLength	:= SIZEOF(wR8604),
	pDestAddr	:= ADR(wR8604));
	PV1	:= WORD_TO_INT(wR8604);

//Motor frequency	
fbR3202(sIPAddr := sIPAddr, nTCPPort := nMBTCPPort, nUnitID := UINT_TO_BYTE(nUnitID), nQuantity := 1, bExecute := bRun, tTimeout := tTimeout,   
	nMBAddr 	:= 3202,
	cbLength	:= SIZEOF(wR3202),
	pDestAddr	:= ADR(wR3202));
	PV2	:= INT_TO_REAL(WORD_TO_INT(wR3202)) / 10;

//Motor current	
fbR3204(sIPAddr := sIPAddr, nTCPPort := nMBTCPPort, nUnitID := UINT_TO_BYTE(nUnitID), nQuantity := 1, bExecute := bRun, tTimeout := tTimeout,   
	nMBAddr 	:= 3204,
	cbLength	:= SIZEOF(wR3204),
	pDestAddr	:= ADR(wR3204));
	PV3	:= INT_TO_REAL(WORD_TO_INT(wR3204)) / 1;

//Motor voltage	
fbR3208(sIPAddr := sIPAddr, nTCPPort := nMBTCPPort, nUnitID := UINT_TO_BYTE(nUnitID), nQuantity := 1, bExecute := bRun, tTimeout := tTimeout,   
	nMBAddr 	:= 3208,
	cbLength	:= SIZEOF(wR3208),
	pDestAddr	:= ADR(wR3208));
	PV4	:= WORD_TO_UINT(wR3208);

//Motor power	
fbR3211(sIPAddr := sIPAddr, nTCPPort := nMBTCPPort, nUnitID := UINT_TO_BYTE(nUnitID), nQuantity := 1, bExecute := bRun, tTimeout := tTimeout,   
	nMBAddr 	:= 3211,
	cbLength	:= SIZEOF(wR3211),
	pDestAddr	:= ADR(wR3211));
	PV7	:= WORD_TO_INT(wR3211);
	
//Drive thermal state	
fbR3209(sIPAddr := sIPAddr, nTCPPort := nMBTCPPort, nUnitID := UINT_TO_BYTE(nUnitID), nQuantity := 1, bExecute := bRun, tTimeout := tTimeout,   
	nMBAddr 	:= 3209,
	cbLength	:= SIZEOF(wR3209),
	pDestAddr	:= ADR(wR3209));
	PV9	:= WORD_TO_INT(wR3209);
	
//Drive state	
fbR3240(sIPAddr := sIPAddr, nTCPPort := nMBTCPPort, nUnitID := UINT_TO_BYTE(nUnitID), nQuantity := 1, bExecute := bRun, tTimeout := tTimeout,   
	nMBAddr 	:= 3240,
	cbLength	:= SIZEOF(wR3240),
	pDestAddr	:= ADR(wR3240));
	
	CASE wR3240 OF 
		0:	PV := 'Autotune';
		1:	PV := 'DC-injektion';
		2:	PV := 'Redo';
		3:	PV := 'Frirullning stopp';
		4:	PV := 'Normaldrift';
		5:	PV := 'Accelererar';
		6:	PV := 'Bromsar';
		7:	PV := 'Strömbegränsning';
		8:	PV := 'Snabbstopp';
		11:	PV := 'Ingen primärspänning';
		13:	PV := 'Kontrollerat stopp';
		14:	PV := 'Nedramp. adaptering';
		15:	PV := 'Klipp utmatning';
		17:	PV := 'Varning underspänning';
		18:	PV := 'TC-läge';
		19:	PV := 'Autotest';
		20:	PV := 'Autotest fel';
		21:	PV := 'Autotest OK';
		22:	PV := 'EEPROM-test';
		23:	PV := 'Driftläge "FAULT"';
		25:	PV := 'DCP-flashläge';
		30:	PV := 'STO aktiv';
		35:	PV := 'Energisparläge';
		36:	PV := 'Firmwareuppdatering';
		37:	PV := 'AFE primär underspänning';
	END_CASE
	
	AL := wR3240 = 23;	//Sätt larmflagga om driftläge FAULT

//Motor thermal state	
fbR9630(sIPAddr := sIPAddr, nTCPPort := nMBTCPPort, nUnitID := UINT_TO_BYTE(nUnitID), nQuantity := 1, bExecute := bRun, tTimeout := tTimeout,   
	nMBAddr 	:= 9630,
	cbLength	:= SIZEOF(wR9630),
	pDestAddr	:= ADR(wR9630));
	PV8	:= WORD_TO_INT(wR9630);	
	
//CiA402 fault code	
fbR8606(sIPAddr := sIPAddr, nTCPPort := nMBTCPPort, nUnitID := UINT_TO_BYTE(nUnitID), nQuantity := 1, bExecute := bRun, tTimeout := tTimeout,   
	nMBAddr 	:= 8606,
	cbLength	:= SIZEOF(wR8606),
	pDestAddr	:= ADR(wR8606));
	PV14	:= wR8606;	

//Last error occurred
fbR7121(sIPAddr := sIPAddr, nTCPPort := nMBTCPPort, nUnitID := UINT_TO_BYTE(nUnitID), nQuantity := 1, bExecute := bRun, tTimeout := tTimeout,   
	nMBAddr 	:= 7121,
	cbLength	:= SIZEOF(wR7121),
	pDestAddr	:= ADR(wR7121));
	PV15	:= wR7121;
	
//Fault counter
fbR7393(sIPAddr := sIPAddr, nTCPPort := nMBTCPPort, nUnitID := UINT_TO_BYTE(nUnitID), nQuantity := 1, bExecute := bRun, tTimeout := tTimeout,   
	nMBAddr 	:= 7393,
	cbLength	:= SIZEOF(wR7393),
	pDestAddr	:= ADR(wR7393));
	PV16	:= wR7393;
	
//Safe torque Off function Status
fbR15322(sIPAddr := sIPAddr, nTCPPort := nMBTCPPort, nUnitID := UINT_TO_BYTE(nUnitID), nQuantity := 1, bExecute := bRun, tTimeout := tTimeout,   
	nMBAddr 	:= 15322,
	cbLength	:= SIZEOF(wR15322),
	pDestAddr	:= ADR(wR15322));
	V3 := wR7393 = 1;
		
//Efficiency
fbR16050(sIPAddr := sIPAddr, nTCPPort := nMBTCPPort, nUnitID := UINT_TO_BYTE(nUnitID), nQuantity := 1, bExecute := bRun, tTimeout := tTimeout,   
	nMBAddr 	:= 16050,
	cbLength	:= SIZEOF(wR16050),
	pDestAddr	:= ADR(wR16050));
	PV11	:= WORD_TO_UINT(wR16050);	
	
//Active Electrical output power estimation
fbR3293(sIPAddr := sIPAddr, nTCPPort := nMBTCPPort, nUnitID := UINT_TO_BYTE(nUnitID), nQuantity := 1, bExecute := bRun, tTimeout := tTimeout,   
	nMBAddr 	:= 3293,
	cbLength	:= SIZEOF(wR3293),
	pDestAddr	:= ADR(wR3293));
	PV5	:= WORD_TO_INT(wR3293);
	
//Number of motor starts
fbR3260_61(sIPAddr := sIPAddr, nTCPPort := nMBTCPPort, nUnitID := UINT_TO_BYTE(nUnitID), bExecute := bRun, tTimeout := tTimeout,
	nQuantity 	:= 2,   
	nMBAddr 	:= 3260,
	cbLength	:= SIZEOF(uR3260_61.aWdata),
	pDestAddr	:= ADR(uR3260_61.aWdata));
	PV13		:= ROR(uR3260_61.ulCombined, 16);

//Input Energy (kWh)
fbR10627(sIPAddr := sIPAddr, nTCPPort := nMBTCPPort, nUnitID := UINT_TO_BYTE(nUnitID), nQuantity := 1, bExecute := bRun, tTimeout := tTimeout,   
	nMBAddr 	:= 10627,
	cbLength	:= SIZEOF(wR10627),
	pDestAddr	:= ADR(wR10627));
	
//Input Energy (MWh)
fbR10628(sIPAddr := sIPAddr, nTCPPort := nMBTCPPort, nUnitID := UINT_TO_BYTE(nUnitID), nQuantity := 1, bExecute := bRun, tTimeout := tTimeout,   
	nMBAddr 	:= 10628,
	cbLength	:= SIZEOF(wR10628),
	pDestAddr	:= ADR(wR10628));
	
//Input Energy (GWh)
fbR10629(sIPAddr := sIPAddr, nTCPPort := nMBTCPPort, nUnitID := UINT_TO_BYTE(nUnitID), nQuantity := 1, bExecute := bRun, tTimeout := tTimeout,   
	nMBAddr 	:= 10629,
	cbLength	:= SIZEOF(wR10629),
	pDestAddr	:= ADR(wR10629));
	
	PV17 := (WORD_TO_DINT(wR10629) * 1000000) + (WORD_TO_DINT(wR10628) * 1000) + WORD_TO_DINT(wR10627);		// Slå ihop GWh+MWh+kWh för att presentera som kWh-räknare	


//Motor mechanical power estimation
fbR3292(sIPAddr := sIPAddr, nTCPPort := nMBTCPPort, nUnitID := UINT_TO_BYTE(nUnitID), nQuantity := 1, bExecute := bRun, tTimeout := tTimeout,   
	nMBAddr 	:= 3292,
	cbLength	:= SIZEOF(wR3292),
	pDestAddr	:= ADR(wR3292));
	PV6	:= WORD_TO_INT(wR3292);	

//Power-on time
fbR3276_77(sIPAddr := sIPAddr, nTCPPort := nMBTCPPort, nUnitID := UINT_TO_BYTE(nUnitID), bExecute := bRun, tTimeout := tTimeout,
	nQuantity 	:= 2,   
	nMBAddr 	:= 3276,
	cbLength	:= SIZEOF(uR3276_77.aWdata),
	pDestAddr	:= ADR(uR3276_77.aWdata));
	PV12		:= ROR(uR3276_77.ulCombined, 16);

//Kom.fel modbus
fbErrorTOF(IN := fbR3201.bError, PT := T#30S);
fbErrorTON(IN := fbErrorTOF.Q, PT := T#180S, Q => AL8);

END_FUNCTION_BLOCK

// oaksModbusLibrary/Server-block/RTU/fbMbRtuSlaveCoilRegBool
//Funktionsblock för COIL register med hantering av BIT in i Word array
FUNCTION_BLOCK fbMbRtuSlaveCoilRegBool
VAR_INPUT
    iReg        : INT; // Register index (Modbus server)
    bRemW       : BOOL; //Värde skrivbart från externt eller inte
END_VAR
VAR_IN_OUT
    bVal        : BOOL;    //Aktuellt värde
END_VAR
VAR
    bInit       : BOOL := TRUE;
    fbInitTimer : TON;
    iBitPos     : INT;
    iWordIndex  : INT;
    iBitMask    : WORD;
	bOldLocVal	: BOOL;
	bOldRemVal	: BOOL;
	wOldVal : WORD;
END_VAR

IF bInit THEN
    fbInitTimer(IN := TRUE, PT := T#5S);
   
    IF fbInitTimer.Q THEN
        bInit := FALSE;
        fbInitTimer(IN := FALSE);
    END_IF
ELSE
    iBitPos := iReg; //Räknar ut bitposition
    iWordIndex := iBitPos / 16; //Räknat ut "Word index" i arrayen
    iBitMask := SHL(1, iBitPos MOD 16); //Skapar bitmask från bitpositon
	
	IF bRemW AND GVL_ModbusRtuSlave.mb_Output[iWordIndex] <> wOldVal THEN
	    wOldVal := GVL_ModbusRtuSlave.mb_Output[iWordIndex];
	    bOldRemVal := WORD_TO_BOOL(wOldVal AND iBitMask); //Tar ut bitvärde
	    bVal := bOldRemVal; //Externt värde
	    bOldLocVal := bVal;
	END_IF
	
	//Lokalt värde ändrat
	IF bVal <> bOldLocVal THEN
	    //Sätter rätt bit i arrayen från lokalt värde
	    IF bVal THEN
	        GVL_ModbusRtuSlave.mb_Output[iWordIndex] := GVL_ModbusRtuSlave.mb_Output[iWordIndex] OR iBitMask;
	    ELSE
	        GVL_ModbusRtuSlave.mb_Output[iWordIndex] := GVL_ModbusRtuSlave.mb_Output[iWordIndex] AND NOT iBitMask;
	    END_IF
	    bOldLocVal := bVal;
	    bOldRemVal := WORD_TO_BOOL(GVL_ModbusRtuSlave.mb_Output[iWordIndex] AND iBitMask);
	END_IF
	
END_IF

END_FUNCTION_BLOCK

// oaksModbusLibrary/Server-block/RTU/fbMbRtuSlaveHoldingRegInt
//Funktionsblock med read/write möjlighet via holding med INT variabel
FUNCTION_BLOCK fbMbRtuSlaveHoldingRegInt
VAR_INPUT
	iReg	: INT;	//Register i array (modbus-server)
	bRemW	: BOOL; //Värde skrivbart från klient/master
END_VAR
VAR_IN_OUT
	iVal	: INT;	//Aktuellt värde
END_VAR
VAR_OUTPUT
END_VAR
VAR
	bInit		: BOOL := 1;
	iOldLocVal	: INT;
	wOldRemVal	: WORD;
	fbInitTimer	: TON;
END_VAR

IF bInit THEN
	fbInitTimer(IN := TRUE, PT := T#5S);
	
	IF fbInitTimer.Q THEN
		bInit := FALSE;
		fbInitTimer(IN := FALSE);
	END_IF
ELSE
	
	IF bRemW AND (GVL_ModbusRtuSlave.mb_Memory[iReg] <> wOldRemVal) THEN		// Fjärrvärde ändrat (om värdet ska kunna ändras utifrån)
		iVal		:= WORD_TO_INT(GVL_ModbusRtuSlave.mb_Memory[iReg]);
		wOldRemVal	:= GVL_ModbusRtuSlave.mb_Memory[iReg];
		iOldLocVal	:= iVal;
	END_IF
	
	IF iVal <> iOldLocVal THEN	// Lokalt värde ändrat
		GVL_ModbusRtuSlave.mb_Memory[iReg] 	:= INT_TO_WORD(iVal);
		iOldLocVal							:= iVal;
		wOldRemVal							:= GVL_ModbusRtuSlave.mb_Memory[iReg];
	END_IF
	
END_IF;

END_FUNCTION_BLOCK

// oaksModbusLibrary/Server-block/RTU/fbMbRtuSlaveHoldingRegReal
//Funktionsblock med read/write möjlighet via holding med REAL variabel
FUNCTION_BLOCK fbMbRtuSlaveHoldingRegReal
VAR_INPUT
	iReg	: INT;	//Register i array (modbus-server)
	iScale	: INT;	//Värde skrivbart från klient/master
	bRemW	: BOOL;
END_VAR
VAR_IN_OUT
	rVal	: REAL;	//Aktuellt värde
END_VAR
VAR_OUTPUT
END_VAR
VAR
	bInit		: BOOL := 1;
	rOldLocVal	: REAL;
	wOldRemVal	: WORD;
	fbInitTimer	: TON;
END_VAR

IF bInit THEN
	fbInitTimer(IN := TRUE, PT := T#5S);
	
	IF fbInitTimer.Q THEN
		bInit := FALSE;
		fbInitTimer(IN := FALSE);
	END_IF
ELSE

	IF iScale < 1 THEN
		iScale := 1;
	END_IF
	
	IF bRemW AND (GVL_ModbusRtuSlave.mb_Memory[iReg] <> wOldRemVal) THEN		// Fjärrvärde ändrat (om värdet ska kunna ändras utifrån)
		rVal		:= INT_TO_REAL(WORD_TO_INT(GVL_ModbusRtuSlave.mb_Memory[iReg])) / iScale;
		wOldRemVal	:= GVL_ModbusRtuSlave.mb_Memory[iReg];
		rOldLocVal	:= rVal;
	END_IF
	
	IF rVal <> rOldLocVal THEN	// Lokalt värde ändrat
		GVL_ModbusRtuSlave.mb_Memory[iReg] 	:= INT_TO_WORD(REAL_TO_INT(rVal * iScale));
		rOldLocVal							:= rVal;
		wOldRemVal							:= GVL_ModbusRtuSlave.mb_Memory[iReg];
	END_IF
	
END_IF;

END_FUNCTION_BLOCK

// oaksModbusLibrary/Server-block/RTU/fbMbRtuSlaveHoldingRegUInt
//Funktionsblock med read/write möjlighet via holding med UINT variabel
FUNCTION_BLOCK fbMbRtuSlaveHoldingRegUInt
VAR_INPUT
	iReg	: INT;	//Register i array (modbus-server)
	bRemW	: BOOL; //Värde skrivbart från klient/master
END_VAR
VAR_IN_OUT
	nVal	: UINT;	//Aktuellt värde
END_VAR
VAR_OUTPUT
END_VAR
VAR
	bInit		: BOOL := 1;
	nOldLocVal	: UINT;
	wOldRemVal	: WORD;
	fbInitTimer	: TON;
END_VAR

IF bInit THEN
	fbInitTimer(IN := TRUE, PT := T#5S);
	
	IF fbInitTimer.Q THEN
		bInit := FALSE;
		fbInitTimer(IN := FALSE);
	END_IF
ELSE
	
	IF bRemW AND (GVL_ModbusRtuSlave.mb_Memory[iReg] <> wOldRemVal) THEN		// Fjärrvärde ändrat (om värdet ska kunna ändras utifrån)
		nVal		:= WORD_TO_UINT(GVL_ModbusRtuSlave.mb_Memory[iReg]);
		wOldRemVal	:= GVL_ModbusRtuSlave.mb_Memory[iReg];
		nOldLocVal	:= nVal;
	END_IF
	
	IF nVal <> nOldLocVal THEN	// Lokalt värde ändrat
		GVL_ModbusRtuSlave.mb_Memory[iReg] 	:= UINT_TO_WORD(nVal);
		nOldLocVal							:= nVal;
		wOldRemVal							:= GVL_ModbusRtuSlave.mb_Memory[iReg];
	END_IF
	
END_IF;

END_FUNCTION_BLOCK

// oaksModbusLibrary/Server-block/RTU/fbMbRtuSlaveStatusRegBool
//Funktionsblock för Status input register med hantering av BIT in i Word array
FUNCTION_BLOCK fbMbRtuSlaveStatusRegBool
VAR_INPUT
    iReg    : INT;  //Register
    bVal    : BOOL; //Värde
END_VAR
VAR
    bInit       : BOOL := TRUE;
    bOldLocVal  : BOOL;
    fbInitTimer : TON;
    iBitPos     : INT;
    iWordIndex  : INT;
    iBitMask    : WORD;
END_VAR

IF bInit THEN
    fbInitTimer(IN := TRUE, PT := T#5S);
    
    IF fbInitTimer.Q THEN
        bInit := FALSE;
        fbInitTimer(IN := FALSE);
    END_IF
ELSE
    iBitPos := iReg MOD 16; //räknar ut bitpotison
    iWordIndex := iReg / 16; //räknar ut word index i arrayen
    iBitMask := SHL(1, iBitPos); //skapar bitmask
    
    //Kollar aktuell status
    bOldLocVal := WORD_TO_BOOL(GVL_ModbusRtuSlave.mb_Input[iWordIndex] AND iBitMask);
    
    //Kollar efter förändring
    IF bVal <> bOldLocVal THEN
        IF bVal THEN
            GVL_ModbusRtuSlave.mb_Input[iWordIndex] := GVL_ModbusRtuSlave.mb_Input[iWordIndex] OR iBitMask;
        ELSE
            GVL_ModbusRtuSlave.mb_Input[iWordIndex] := GVL_ModbusRtuSlave.mb_Input[iWordIndex] AND NOT iBitMask;
        END_IF
    END_IF
END_IF;

END_FUNCTION_BLOCK

// oaksModbusLibrary/Server-block/fbMbSlaveRegBool
//Mappning av bool-variabler till Modbus Server i TC3, för både läsning och skrivning eller endast läsning (bRemW false)
//OBS! Förutsätter att arrayen mb_Coils finns i GVL ModbusServer (se mall för Modbus Server/Slave)

FUNCTION_BLOCK fbMbSlaveRegBool
VAR_INPUT
	iReg	: INT;		//Register i array (modbus-server)
	bRemW	: BOOL;		//Värde skrivbart från klient/master
END_VAR
VAR_IN_OUT
	bVal	: BOOL;		//Aktuellt värde
END_VAR
VAR_OUTPUT
END_VAR
VAR
	bInit		: BOOL := 1;
	bOldLocVal	: BOOL;
	bOldRemVal	: BOOL;
	fbInitTimer	: TON;
END_VAR

IF bInit THEN
	fbInitTimer(IN := TRUE, PT := T#5S);
	
	IF fbInitTimer.Q THEN
		bInit := FALSE;
		fbInitTimer(IN := FALSE);
	END_IF
ELSE
	
	IF ModbusServer.mb_Coils[iReg] <> bOldRemVal THEN		// Fjärrvärde ändrat
		bVal		:= ModbusServer.mb_Coils[iReg];
		bOldRemVal	:= bVal;
		bOldLocVal	:= bVal;
	END_IF
	
	IF bVal <> bOldLocVal THEN	// Lokalt värde ändrat
		ModbusServer.mb_Coils[iReg]			:= bVal;
		bOldLocVal							:= bVal;
		bOldRemVal							:= ModbusServer.mb_Coils[iReg];
	END_IF
	
END_IF;

END_FUNCTION_BLOCK

// oaksModbusLibrary/Server-block/fbMbSlaveRegInt
//Mappning av INT-variabler till Modbus Server i TC3, för både läsning och skrivning eller endast läsning (bRemW false)
//OBS! Förutsätter att arrayen mb_HoldingRegs finns i GVL ModbusServer (se mall för Modbus Server/Slave)

FUNCTION_BLOCK fbMbSlaveRegInt
VAR_INPUT
	iReg	: INT;	//Register i array (modbus-server)
	bRemW	: BOOL;	//Värde skrivbart från klient/master
END_VAR
VAR_IN_OUT
	iVal	: INT;	//Aktuellt värde
END_VAR
VAR_OUTPUT
END_VAR
VAR
	bInit		: BOOL := 1;
	iOldLocVal	: REAL;
	wOldRemVal	: WORD;
	fbInitTimer	: TON;
END_VAR

IF bInit THEN
	fbInitTimer(IN := TRUE, PT := T#5S);
	
	IF fbInitTimer.Q THEN
		bInit := FALSE;
		fbInitTimer(IN := FALSE);
	END_IF
ELSE
	
	IF bRemW AND (ModbusServer.mb_HoldingRegs[iReg] <> wOldRemVal) THEN		// Fjärrvärde ändrat (om värdet ska kunna ändras utifrån)
		iVal		:= WORD_TO_INT(ModbusServer.mb_HoldingRegs[iReg]);
		wOldRemVal	:= ModbusServer.mb_HoldingRegs[iReg];
		iOldLocVal	:= iVal;
	END_IF
	
	IF iVal <> iOldLocVal THEN	// Lokalt värde ändrat
		ModbusServer.mb_HoldingRegs[iReg] 	:= INT_TO_WORD(iVal);
		iOldLocVal							:= iVal;
		wOldRemVal							:= ModbusServer.mb_HoldingRegs[iReg];
	END_IF
	
END_IF;

END_FUNCTION_BLOCK

// oaksModbusLibrary/Server-block/fbMbSlaveRegReal
//Mappning av REAL-variabler till Modbus Server i TC3, för både läsning och skrivning eller endast läsning (bRemW false)
//OBS! Förutsätter att arrayen mb_HoldingRegs finns i GVL ModbusServer (se mall för Modbus Server/Slave)

FUNCTION_BLOCK fbMbSlaveRegReal
VAR_INPUT
	iReg	: INT;	//Register i array (modbus-server)
	iScale	: INT;	//Värde skrivbart från klient/master
	bRemW	: BOOL;
END_VAR
VAR_IN_OUT
	rVal	: REAL;	//Aktuellt värde
END_VAR
VAR_OUTPUT
END_VAR
VAR
	bInit		: BOOL := 1;
	rOldLocVal	: REAL;
	wOldRemVal	: WORD;
	fbInitTimer	: TON;
END_VAR

IF bInit THEN
	fbInitTimer(IN := TRUE, PT := T#5S);
	
	IF fbInitTimer.Q THEN
		bInit := FALSE;
		fbInitTimer(IN := FALSE);
	END_IF
ELSE

	IF iScale < 1 THEN
		iScale := 1;
	END_IF
	
	IF bRemW AND (ModbusServer.mb_HoldingRegs[iReg] <> wOldRemVal) THEN		// Fjärrvärde ändrat (om värdet ska kunna ändras utifrån)
		rVal		:= INT_TO_REAL(WORD_TO_INT(ModbusServer.mb_HoldingRegs[iReg])) / iScale;
		wOldRemVal	:= ModbusServer.mb_HoldingRegs[iReg];
		rOldLocVal	:= rVal;
	END_IF
	
	IF rVal <> rOldLocVal THEN	// Lokalt värde ändrat
		ModbusServer.mb_HoldingRegs[iReg] 	:= INT_TO_WORD(REAL_TO_INT(rVal * iScale));
		rOldLocVal							:= rVal;
		wOldRemVal							:= ModbusServer.mb_HoldingRegs[iReg];
	END_IF
	
END_IF;

END_FUNCTION_BLOCK

// oaksModbusLibrary/Server-block/fbMbSlaveRegUInt
//Mappning av UINT-variabler till Modbus Server i TC3, för både läsning och skrivning eller endast läsning (bRemW false)
//OBS! Förutsätter att arrayen mb_HoldingRegs finns i GVL ModbusServer (se mall för Modbus Server/Slave)

FUNCTION_BLOCK fbMbSlaveRegUInt
VAR_INPUT
	iReg	: INT;	//Register i array (modbus-server)
	bRemW	: BOOL;	//Värde skrivbart från klient/master
END_VAR
VAR_IN_OUT
	nVal	: UINT;	//Aktuellt värde
END_VAR
VAR_OUTPUT
END_VAR
VAR
	bInit		: BOOL := 1;
	nOldLocVal	: UINT;
	wOldRemVal	: WORD;
	fbInitTimer	: TON;
END_VAR

IF bInit THEN
	fbInitTimer(IN := TRUE, PT := T#5S);
	
	IF fbInitTimer.Q THEN
		bInit := FALSE;
		fbInitTimer(IN := FALSE);
	END_IF
ELSE
	
	IF bRemW AND (ModbusServer.mb_HoldingRegs[iReg] <> wOldRemVal) THEN		// Fjärrvärde ändrat (om värdet ska kunna ändras utifrån)
		nVal		:= WORD_TO_INT(ModbusServer.mb_HoldingRegs[iReg]);
		wOldRemVal	:= ModbusServer.mb_HoldingRegs[iReg];
		nOldLocVal	:= nVal;
	END_IF
	
	IF nVal <> nOldLocVal THEN	// Lokalt värde ändrat
		ModbusServer.mb_HoldingRegs[iReg] 	:= INT_TO_WORD(nVal);
		nOldLocVal							:= nVal;
		wOldRemVal							:= ModbusServer.mb_HoldingRegs[iReg];
	END_IF
	
END_IF;

END_FUNCTION_BLOCK

// oaksModbusLibrary/Siemens/Spjäll/fbSiemensGDB1811EMO
//OAKS AB
//2020-11-16
//Funktionsblock för modbus-TCP, Siemens GDB181.1E-MO. Spjäll konfigureras via block till mätning i l/s (register 389) samt styrning som VAV (register 259).
//Används i VAV-läge med l/s.
//Uträkning av börvärde finns ej inbyggt utan sker i PLC. (endast då själl står i auto iMode=0). 
FUNCTION_BLOCK fbSiemensGDB1811EMO
VAR_INPUT
	sIPAddr : STRING := ''; 
	nTCPPort : UINT;
	nUnitID : UINT :=1;
	iModbusLoop : INT :=1; //Modbusslinga
	rSetpoint : REAL; //Börvärde
	iMode : INT; //Överstyrning spjäll-läge 0: None 1: Open 2: Close 3: Min 4: Mid 5: MAX
	SP1 AT %M* : REAL;//Min-flöde~wp:[unit]%[format]0[trendoptions]i:300
	SP2 AT %M* : REAL;//Max-flöde~wp:[unit]%[format]0[trendoptions]i:300	
		
END_VAR
VAR_OUTPUT
	
	PV1 AT %M* : REAL;//Volym~wp:[unit]l/s[format]0[trendoptions]i:300
	PV4 AT %M* : REAL;//Aktuellt diff.tryck~wp:[unit]Pa[format]0[trendoptions]i:300
	PV5 AT %M* : UINT;//Spjäll-läge 0: None 1: Open 2: Close 3: Min 4: Mid 5: MAX~wp:[format]0[trendoptions]i:14400, t:1
	PV6 AT %M* : UINT;//Nominellt volym flöde~wp:[unit]l/s[format]0[trendoptions]i:300
	PV7 AT %M* : REAL;//Inställt min-flöde~wp:[unit]l/s[format]0[trendoptions]i:300
	PV8 AT %M* : REAL;//Inställt max-flöde~wp:[unit]l/s[format]0[trendoptions]i:300
	PV9 AT %M* : REAL;//Inställt min-flöde~wp:[unit]%[format]0[trendoptions]i:300
	PV10 AT %M* : REAL;//Inställt max-flöde~wp:[unit]%[format]0[trendoptions]i:300
	PV11 AT %M* : STRING;//Modbus konfigurering~wp:
	CSP AT %M* : REAL;//Uträknat börvärde~wp:[unit]l/s[format]0[trendoptions]i:300
	OP AT %M* : REAL;//Relativ position~wp:[unit]%[format]0[trendoptions]i:300	
	FAULT AT %M* : BOOL;//Kommunikationsfel~wp:
	AL AT %M* : BOOL;//Driftfel spjäll~wp:
	
END_VAR
VAR
	rTemp : REAL;
	iTemp : UINT;
	wTemp : WORD;
	bSekvensFlagga : BOOL;
	
	FB_MBReadRegs_ArrHolding1: FB_MBReadRegs;
	wArrHolding1 : ARRAY [1..6] OF WORD; //Holding
	wActSetpoint : WORD; //Börvärde 0
	wModeOut : WORD; //Överstyrning 1 
	wActualPos : WORD; //Relativ position 2
	wAbsVolume : WORD; //Volym 4
	wdiffPress: WORD; //Diff.press 5

	FB_MBReadRegs_ArrHolding2 : FB_MBReadRegs;
	wArrHolding2 : ARRAY [257..262] OF WORD; //Holding	
	wOpMode : WORD; //Operating mode 259 
		
	FB_MBReadRegs_ArrHolding3 : FB_MBReadRegs;
	wArrHolding3 : ARRAY [385..389] OF WORD; //Holding	
	wVmin : WORD; //Min setpoint 105
	wVmax : WORD; //Max setpoint 106
	wNomVolFlow : WORD; //Nominellt volym flöde l/s
	wUnitSwitch: WORD;
	
	FB_MBReadRegs_ArrHoldingAlarm: FB_MBReadRegs;
	wAlarm : WORD; //Fel 769
	
	//Skrivning
	FB_MBWriteSingleReg_OperatingMode: FB_MBWriteSingleReg;
	
	FB_MBWriteSingleReg_UnitSwitch: FB_MBWriteSingleReg;
	
	FB_MBWriteSingleReg_Setpoint : FB_MBWriteSingleReg; 
	FB_MBWriteSingleReg_Mode : FB_MBWriteSingleReg; 
		
	fbWriteHoldingDoubleControlledMin: fbDoubleControlledModbusHolding;
	fbWriteHoldingDoubleControlledMax: fbDoubleControlledModbusHolding;
	
	//Kommunikationsfel
	fbKommTof : tof;
	fbAlarm_ComError: fbAlarm; 
			
	sIP: STRING(255);
	sPort: STRING(255);
	sModbusID: STRING(255);
	sModbusLoop: STRING(255);
	sTemp : STRING(255);
		
	fbAlarm_Alarm: fbAlarm;
	
	fb_CSP : Tc3_BA.FB_BA_Chrct02;
		
END_VAR

VAR_IN_OUT

END_VAR

//Offset satt till -1

//Sekvens
	bSekvensFlagga := oaksGVL.aBModbusSekvens[iModbusLoop] = UINT_TO_INT(nUnitID);
//Modbus konfiguering
	sIP := CONCAT (SIPAddr, '');
	sPort := CONCAT ('<br>Port: ', UINT_TO_STRING(nTCPPort)); 								
	sModbusID := CONCAT('<br>ID: ', UINT_TO_STRING(nUnitID));
	sModbusLoop := CONCAT('<br>Loop: ', INT_TO_STRING(iModbusLoop));	

	sTemp := sIP;
	sTemp := CONCAT(sTemp, sPort);
	sTemp := CONCAT(sTemp, sModbusID);
	sTemp := CONCAT(sTemp, sModbusLoop);
	
	PV11 := sTemp;
 
///////////////		
//READ
///////////////		
	
	//Read Holding 0-5
	FB_MBReadRegs_ArrHolding1(
	sIPAddr:= sIpAddr, 
	nTCPPort:= INT_TO_UINT(nTCPPort), 
	nUnitID:= INT_TO_BYTE(nUnitID), 
	nQuantity:= 6, 
	nMBAddr:= 0, 
	cbLength:= SIZEOF(wArrHolding1), 
	pDestAddr:= ADR(wArrHolding1), 
	bExecute:= bSekvensFlagga, 
	tTimeout:= T#3S, 
	bBusy=> , 
	bError=> , 
	nErrId=> , 
	cbRead=> );
	
		//Values
		wActSetpoint := wArrHolding1[1]; //1
		wModeOut := wArrHolding1[2]; //2
		wActualPos := wArrHolding1[3]; //3
		//wArrHolding1[4]; //4
		wAbsVolume := wArrHolding1[5]; //5
		wdiffPress := wArrHolding1[6]; //6
						
		//Absolute Volume flow
		PV1 := wAbsVolume;
	
		//Actual Position
		
		iTemp := WORD_TO_UINT(wActualPos);
		rTemp := UINT_TO_REAL(iTemp);
		OP := rTemp / 100;
		
		//Actual diff.press
		iTemp := WORD_TO_UINT(wdiffPress);
		rTemp := UINT_TO_REAL(iTemp);
		PV4 := rTemp / 10;
				
		//Actual damper-mode
		PV5 := WORD_TO_UINT(wModeOut);

	//Read Holding 257-262
	FB_MBReadRegs_ArrHolding2(
	sIPAddr:= sIpAddr, 
	nTCPPort:= INT_TO_UINT(nTCPPort), 
	nUnitID:= INT_TO_BYTE(nUnitID), 
	nQuantity:= 6, 
	nMBAddr:= 256, 
	cbLength:= SIZEOF(wArrHolding2), 
	pDestAddr:= ADR(wArrHolding2), 
	bExecute:= bSekvensFlagga, 
	tTimeout:= T#3S, 
	bBusy=> , 
	bError=> , 
	nErrId=> , 
	cbRead=> );
	
		//Tilldela värden
		//wArrHolding2[257];
		//wArrHolding2[258];
		wOpMode := wArrHolding2[259];
		//wArrHolding2[260];
		//wArrHolding2[261];
		//wArrHolding2[262];
						
	//Read Holding 385-389
	FB_MBReadRegs_ArrHolding3(
	sIPAddr:= sIpAddr, 
	nTCPPort:= INT_TO_UINT(nTCPPort), 
	nUnitID:= INT_TO_BYTE(nUnitID), 
	nQuantity:= 5, 
	nMBAddr:= 384, 
	cbLength:= SIZEOF(wArrHolding3), 
	pDestAddr:= ADR(wArrHolding3), 
	bExecute:= bSekvensFlagga, 
	tTimeout:= T#3S, 
	bBusy=> , 
	bError=> , 
	nErrId=> , 
	cbRead=> );
	
		//Tilldela värden
		wNomVolFlow := wArrHolding3[385]; //385
		wVmin := wArrHolding3[386]; //386
		wVmax := wArrHolding3[387]; //387
		//wArrHolding3[388]; //388
		wUnitSwitch := wArrHolding3[389]; //389
			
		//Nominal Volume flow (m2/h)
		PV6 := wNomVolFlow;
					
		//Setpoint min-flow 
		iTemp := WORD_TO_UINT(wVmin);
		rTemp := fSignedConverter(UINT_TO_REAL(iTemp));
		PV7 :=  (rTemp /10000) * wNomVolFlow;
		PV9 :=  (rTemp /100);		
				
		//Setpoint max-flow 
		iTemp := WORD_TO_UINT(wVmax);
		rTemp := fSignedConverter(UINT_TO_REAL(iTemp));	
			
		PV8 :=  (rTemp /10000) * wNomVolFlow;
		PV10 := (rTemp /100);
		
	//Alarm
	//Read Holding 769
	FB_MBReadRegs_ArrHoldingAlarm(
	sIPAddr:= sIpAddr, 
	nTCPPort:= INT_TO_UINT(nTCPPort), 
	nUnitID:= INT_TO_BYTE(nUnitID), 
	nQuantity:= 1, 
	nMBAddr:= 768, 
	cbLength:= SIZEOF(wAlarm), 
	pDestAddr:= ADR(wAlarm), 
	bExecute:= bSekvensFlagga, 
	tTimeout:= T#3S, 
	bBusy=> , 
	bError=> , 
	nErrId=> , 
	cbRead=> );	

	fbAlarm_Alarm(bInput:= wAlarm.0 OR wAlarm.1 OR wAlarm.2 OR wAlarm.3 OR wAlarm.4 OR wAlarm.8 OR wAlarm.9 OR wAlarm.11, tAlarmDelay:= T#1M, bAutoReset:= TRUE, bAlarmOutput=> AL);
				
///////////////		
//WRITE
///////////////	

//Operating mode
		
	IF 0 <> wOpMode AND bSekvensFlagga THEN
		FB_MBWriteSingleReg_OperatingMode.bExecute := TRUE;
	ELSE
		FB_MBWriteSingleReg_OperatingMode.bExecute := FALSE;
		
	END_IF
	
	//Write Operating mode
	FB_MBWriteSingleReg_OperatingMode(
	sIPAddr:= sIpAddr, 
	nTCPPort:= INT_TO_UINT(nTCPPort), 
	nUnitID:= INT_TO_BYTE(nUnitID), 
	nMBAddr:= 258, 
	nValue:= 0, 
	bExecute:= , 
	tTimeout:= T#3S, 
	bBusy=> , 
	bError=> , 
	nErrId=> );

//Unit Switch (Sätt mätning till l/s)
		
	IF 1 <> wUnitSwitch AND bSekvensFlagga THEN
		FB_MBWriteSingleReg_UnitSwitch.bExecute := TRUE;
	ELSE
		FB_MBWriteSingleReg_UnitSwitch.bExecute := FALSE;
		
	END_IF
	
	//Write UnitSwitch
	FB_MBWriteSingleReg_UnitSwitch(
	sIPAddr:= sIpAddr, 
	nTCPPort:= INT_TO_UINT(nTCPPort), 
	nUnitID:= INT_TO_BYTE(nUnitID), 
	nMBAddr:= 388, 
	nValue:= 1, 
	bExecute:= , 
	tTimeout:= T#3S, 
	bBusy=> , 
	bError=> , 
	nErrId=> );
				
//Setpoint
	rTemp := LIMIT (0, rSetpoint, 100);
	wTemp := frealtoword(rTemp, 100);
	
	IF wTemp <> wActSetpoint AND bSekvensFlagga THEN
		FB_MBWriteSingleReg_Setpoint.bExecute := TRUE;
	ELSE
		FB_MBWriteSingleReg_Setpoint.bExecute := FALSE;
		
	END_IF
	
	//Write Setpoint
	FB_MBWriteSingleReg_Setpoint(
	sIPAddr:= sIpAddr, 
	nTCPPort:= INT_TO_UINT(nTCPPort), 
	nUnitID:= INT_TO_BYTE(nUnitID), 
	nMBAddr:= 0, 
	nValue:= wTemp, 
	bExecute:= , 
	tTimeout:= T#3S, 
	bBusy=> , 
	bError=> , 
	nErrId=> );
	
//Override

	iTemp := INT_TO_WORD(iMode);	
	
	IF wModeOut <> iTemp AND bSekvensFlagga THEN 
		FB_MBWriteSingleReg_Mode.bExecute := TRUE;
	ELSE 
		FB_MBWriteSingleReg_Mode.bExecute := FALSE;
	END_IF
	
	//Write Mode
	FB_MBWriteSingleReg_Mode(
	sIPAddr:= sIpAddr, 
	nTCPPort:= INT_TO_UINT(nTCPPort), 
	nUnitID:= INT_TO_BYTE(nUnitID), 
	nMBAddr:= 1, 
	nValue:= UINT_TO_WORD(iTemp), 
	bExecute:= , 
	tTimeout:= T#3S, 
	bBusy=> , 
	bError=> , 
	nErrId=> );

//Read/write

//Min
	fbWriteHoldingDoubleControlledMin(
	sIPAddr:= sIPAddr, 
	nTCPPort:= nTCPPort, 
	nUnitID:= UINT_TO_BYTE(nUnitID) , 
	nMBAddr:= 385, 
	bExecute:= bSekvensFlagga, 
	rScale:= 100, 
	rWrite:= SP1, 
	bBusy=> , 
	bError=> );
//Max		
	fbWriteHoldingDoubleControlledMax(
	sIPAddr:= sIPAddr, 
	nTCPPort:= nTCPPort, 
	nUnitID:= UINT_TO_BYTE(nUnitID) , 
	nMBAddr:= 386, 
	bExecute:= bSekvensFlagga, 
	rScale:= 100, 
	rWrite:= SP2, 
	bBusy=> , 
	bError=> );
	
//Communication error
	fbKommTof(IN:=FB_MBReadRegs_ArrHolding1.bError OR FB_MBReadRegs_Arrholding2.bError OR FB_MBReadRegs_Arrholding3.bError OR FB_MBReadRegs_ArrHoldingAlarm.bError, PT:=T#20S , Q=> , ET=> );
	fbAlarm_ComError(bInput:= fbKommTof.Q, tAlarmDelay:= T#20M, bAutoReset:= TRUE, bAlarmOutput=> FAULT);
		
//Write busy	
	oaksgvl.aBModbusBusyFlagga[iModbusLoop,nUnitID] := FB_MBReadRegs_Arrholding1.bBusy OR FB_MBReadRegs_Arrholding2.bBusy OR FB_MBReadRegs_Arrholding3.bBusy OR FB_MBReadRegs_ArrHoldingAlarm.bBusy OR 
	FB_MBWriteSingleReg_OperatingMode.bBusy OR FB_MBWriteSingleReg_UnitSwitch.bBusy OR FB_MBWriteSingleReg_Setpoint.bBusy OR FB_MBWriteSingleReg_Mode.bBusy OR fbWriteHoldingDoubleControlledMin.bBusy OR fbWriteHoldingDoubleControlledMax.bBusy;
	
//Calculated setpoint
	fb_CSP(
	rX:= WORD_TO_REAL(wActSetpoint) / 100, 
	rX01:= 0, 
	rX02:= 100, 
	rY01:= PV7, 
	rY02:= PV8, 
	bLmt:= TRUE, 
	rY=> , 
	bErr=> , 
	sErrDescr=> );

	IF wOpMode = 0 THEN
		CSP := fb_CSP.rY;
	ELSE 
		CSP := 0;
	END_IF

END_FUNCTION_BLOCK

// oaksModbusLibrary/Siox/Via modul/fbSioxDamperDUOdirect
//OAKS AB
//2022-03-17
//Funktionsblock för kommunikation med direkt med SIOX-DUO spjällmodul (2st spläll).
//Läser transparent genom SX:access enhet. Krävs att register holding register 63 sätts till 1 i SX:Access.
//Läsning via adress 1-59. Aktuell SIOX-adress är samma som Modbus-ID.

//För att aktivera kommando del krävs aktivering via bEnableMan
//För att aktivera skrivning till analog utgång aktivering via bSetpointDamperXEnable
FUNCTION_BLOCK fbSioxDamperDUOdirect EXTENDS fbSioxDamperUNOdirect

VAR_INPUT
	bSetpointDamper2Enable : BOOL; // Aktivera skrivning av 0-10V signal
	rSetpointDamper2 : REAL; // Värde 0-10V signal (0-100 skalning)
END_VAR
VAR_OUTPUT
	DAMPER2_AL  AT %M*  : BOOL; //Driftfel spjäll 2~wp:
	DAMPER2_V0  AT %M*  : BOOL; //Stängtindikering spjäll 2~wp:[trendoptions]i:14400, t:1
	DAMPER2_V1  AT %M*  : BOOL; //Öppetindikering spjäll 2~wp:[trendoptions]i:14400, t:1
END_VAR
VAR

	rSetpointDamper1Internal2: REAL;
END_VAR

SUPER^();
//Modbus konfiguering
	DAMPER2_AL := wInternalWord.5;
	DAMPER2_V0 := wInternalWord.10;
	DAMPER2_V1 := wInternalWord.11;
	
	//Begränsa insignal 0-100%
	rSetpointDamper1Internal2 := LIMIT(0,rSetpointDamper2,100);
	
	//Skriv utsignal
	fbReadWriteHoldingRegDamper2(
	sIPAddr:= modbusTCP.sIPAddr, 
	nTCPPort:= modbusTCP.nTCPPort, 
	nUnitID:= nUnitID, 
	mBusAdr:=7 , 
	bEnable:= bSetpointDamper2Enable AND bSekvensFlagga, 
	tTimeout:= T#5S, 
	rReal:= fScale2pInternalSetpoint(rX:=rSetpointDamper1Internal2 , Y1:=0 , Y2:=4096 , X1:=0 , X2:=100 ), 
	uiFaktor:= 1, 
	bError=> , 
	bBusy=> );

END_FUNCTION_BLOCK

// oaksModbusLibrary/Siox/Via modul/fbSioxDamperUNOdirect
//OAKS AB
//2022-03-17
//Funktionsblock för kommunikation med direkt med SIOX-UNO spjällmodul (1st spläll).
//Läser transparent genom SX:access enhet. Krävs att register holding register 63 sätts till 1 i SX:Access.
//Läsning via adress 1-59. Aktuell SIOX-adress är samma som Modbus-ID.

//För att aktivera kommandodel krävs aktivering via bEnableCommand
//För att aktivera skrivning till analog utgång aktivering via bSetpointDamperXEnable
FUNCTION_BLOCK fbSioxDamperUNOdirect

VAR_INPUT
	modbusTCP : ST_ModbusTCP := (sIPAddr:='127.1.1.0', nTCPPort:=502, iModbusLoop:=1);
	nUnitID : BYTE := 1; //Modbus-ID/SIOX-adr 1-59
	bSetpointDamper1Enable : BOOL; // Aktivera skrivning av 0-10V signal
	rSetpointDamper1 : REAL;// Värde 0-10V signal (0-100 skalning)
	//Manöver
	bEnableCommand : BOOL := FALSE; //Aktivera manöver
	bCloseDampers : BOOL := FALSE; //Stäng spjäll (True=stäng spjäll)
	bExerciseOnRisingTrig : BOOL := FALSE;
END_VAR
VAR_OUTPUT
	V AT %M*  : BOOL; //Standby bit (1=Standby)~wp:[trendoptions]i:14400, t:1
	PV5 AT %M*  : BOOL; //Motionskörning~wp:[trendoptions]i:14400, t:1
	AL AT %M*  : BOOL; //Övertemperatur (NTC)~wp:
	FAULT AT %M*  : BOOL; //Kommunikationsfel Siox~wp:
	GX_V  AT %M*  : BOOL; //Rökdetektor I drift~wp:[trendoptions]i:14400, t:1
	GX_AL  AT %M*  : BOOL; //Utlöst rökdetektor~wp:
	GX_AL1  AT %M*  : BOOL;  //Servicelarm rökdetektor~wp:
	GX_AL2  AT %M*  : BOOL; //Slingfel~wp:
	PV8 AT %M* : STRING;//Modbus konfiguering~wp:
	DAMPER1_AL  AT %M*  : BOOL; //Driftfel spjäll 1~wp:  
	DAMPER1_V0  AT %M*  : BOOL; //Stängtindikering spjäll 1~wp:[trendoptions]i:14400, t:1
	DAMPER1_V1  AT %M*  : BOOL; //Öppetindikering spjäll 1~wp:[trendoptions]i:14400, t:1
END_VAR
VAR
	RST AT %M*  : BOOL := FALSE; //Återställning lokala larm (UNO)~wp:
	M AT %M*  : BOOL := FALSE; //Funktionstest/motionering (UNO)~wp:[trendoptions]i:14400, t:1
	rTemp : REAL;
	iTemp : UINT;
	bSekvensFlagga : BOOL;	

	wInternalWord : WORD;
	fbKommTof: Tof;
	fbKommTon: Ton;
	FB_MBReadRegs01: FB_MBReadRegs;
	fbtoggle1 : fbToggle;
	
	sIP: STRING(255);
	sPort: STRING(255);
	sModbusID: STRING(255);
	sModbusLoop: STRING(255);
	sTemp : STRING(255);
	sTemp1 : STRING(255);
	wTemp : WORD;
	fbReadWriteHoldingRegDamper1: fbReadWriteHoldingRegReal;
	fbReadWriteHoldingRegDamper2: fbReadWriteHoldingRegReal;
	fbReadWriteHoldingRegManover: fbReadWriteHoldingRegReal;
	
	//Manöver
	rManover : WORD;
	R_TRIG_Motion: F_TRIG;
	R_TRIG_Reset: F_TRIG;
	
	rSetpointDamper1Internal1: REAL;
	
	
	rTrigExercise : R_TRIG;
	bExercise : BOOL;
END_VAR

//Sekvens	
	bSekvensFlagga := oaksGVL.aBModbusSekvens[modbusTCP.iModbusLoop]= nUnitID;

	//Begränsa insignal 0-100%
	rSetpointDamper1Internal1 := LIMIT(0,rSetpointDamper1,100);
	
	//Skriv utsignal
	fbReadWriteHoldingRegDamper1(
	sIPAddr:= modbusTCP.sIPAddr, 
	nTCPPort:= modbusTCP.nTCPPort, 
	nUnitID:= nUnitID , 
	mBusAdr:=6 , 
	bEnable:= bSetpointDamper1Enable AND bSekvensFlagga, 
	tTimeout:= T#5S, 
	rReal:= fScale2pInternalSetpoint(rX:=rSetpointDamper1Internal1 , Y1:=0 , Y2:=4096 , X1:=0 , X2:=100 ), 
	uiFaktor:= 1, 
	bError=> , 
	bBusy=> );
	
//Manöver
	rManover.0 := FALSE; //Forced damper opening
	rManover.1 := FALSE; //External firealarm
	rManover.2 := RST;//Reset local alarms
	rManover.3 := bCloseDampers; //Close dampers
	rManover.4 := M OR bExercise; //Function test / Excersise
	rManover.5 := FALSE;
	rManover.6 := FALSE;
	rManover.7 := FALSE;
	rManover.8 := FALSE;
	rManover.9 := FALSE;
	rManover.10 := FALSE;
	rManover.11 := FALSE;
	rManover.12 := FALSE;
	rManover.13 := FALSE;
	rManover.14 := FALSE;
	rManover.15 := FALSE;
	
	//Skriv
	fbReadWriteHoldingRegManover(
	sIPAddr:= modbusTCP.sIPAddr, 
	nTCPPort:= modbusTCP.nTCPPort, 
	nUnitID:= nUnitID, 
	mBusAdr:=44 , 
	bEnable:= bSekvensFlagga AND bEnableCommand,
	tTimeout:= T#5S, 
	rReal:= rManover, 
	uiFaktor:= 1, 
	bError=> , 
	bBusy=> ); 
	
	//Kör endast en gång via ingång och tills dess att skrivning är ok
	rTrigExercise(CLK:=bExerciseOnRisingTrig , Q=>);
	
	IF rTrigExercise.Q THEN
		bExercise := TRUE;
	END_IF
	
	//Återställ motion om skrivning gick igenom
	R_TRIG_Motion(CLK:= fbReadWriteHoldingRegManover.bSuccess, Q=> );
	
	IF R_TRIG_Motion.Q THEN
		M := FALSE;
		bExercise := FALSE;
	END_IF
	
	R_TRIG_Reset(CLK:= fbReadWriteHoldingRegManover.bSuccess, Q=> );
	
	IF R_TRIG_Reset.Q THEN
		RST := FALSE;
	END_IF

//Modbus konfiguering
	sIP := CONCAT (modbusTCP.sIPAddr, '');
	sPort := CONCAT ('<br>Port: ', UINT_TO_STRING(modbusTCP.nTCPPort));
	sModbusID := CONCAT('<br>Modbus-ID/SIOX-adr: ', UINT_TO_STRING(nUnitID));
	sModbusLoop := CONCAT('<br>Loop: ', INT_TO_STRING(modbusTCP.iModbusLoop));

	sTemp := sIP;
	sTemp := CONCAT(sTemp, sPort);
	sTemp := CONCAT(sTemp, sModbusID);
	sTemp := CONCAT(sTemp, sModbusLoop);
	
	PV8 := sTemp;
		
FB_MBReadRegs01(
	sIPAddr:= modbusTCP.sIPAddr, 
	nTCPPort:= modbusTCP.nTCPPort, 
	nUnitID:= nUnitID, 
	nQuantity:= 1, 
	nMBAddr:= 32, 
	cbLength:= SIZEOF(wInternalWord), 
	pDestAddr:=ADR(wInternalWord) , 
	bExecute:=bSekvensFlagga , 
	tTimeout:=T#4S , 
	bBusy=> , 
	bError=> , 
	nErrId=> , 
	cbRead=> );
	
	V := wInternalWord.0;
	PV5 := wInternalWord.4;
	AL :=  wInternalWord.7;
	DAMPER1_AL := wInternalWord.3;
	DAMPER1_V0 := wInternalWord.8;
	DAMPER1_V1 := wInternalWord.9;
	(* Används i DUO
	DAMPER2_AL := wInternalWord.5;
	DAMPER2_V0 := wInternalWord.10;
	DAMPER2_V1 := wInternalWord.11;
	*)
	GX_AL := wInternalWord.13;
	GX_AL1 := wInternalWord.14;
	GX_AL2 := wInternalWord.15;
	GX_V := wInternalWord.12;
	
	//Communication error
	fbKommTof(IN:=FB_MBReadRegs01.bError , PT:=T#20S , Q=> , ET=> );
	fbKommTon(IN:=fbKommTof.Q , PT:=T#20M , Q=> , ET=> );
	FAULT :=fbKommTon.Q;
		
//Write busy	
	oaksgvl.aBModbusBusyFlagga[modbusTCP.iModbusLoop,nUnitID] := FB_MBReadRegs01.bBusy OR fbReadWriteHoldingRegDamper1.bBusy OR fbReadWriteHoldingRegDamper2.bBusy OR fbReadWriteHoldingRegManover.bBusy;

END_FUNCTION_BLOCK

// oaksModbusLibrary/Siox/Via modul/fbSioxSxAcura
//OAKS AB
//2022-10-26
//Modbusblock för avläsning och styrning av SIOX SX:ACURA (2AI/2AO)
FUNCTION_BLOCK fbSioxSxAcura
VAR_INPUT
	bEnable			: BOOL;
	modbusTCP		: ST_ModbusTCP 	:= (sIPAddr:='127.1.1.0', nTCPPort:=502, iModbusLoop:=1);
	nUnitID 		: BYTE := 1; //Modbus-ID/SIOX-adr 1-59
	rSetpointAO1 	: REAL :=0; //Värde 0-10V signal (0-100 skalning)
	rSetpointAO2	: REAL :=0; //Värde 0-10V signal (0-100 skalning)
	rScaleAI1min 	: REAL :=0; //Min-värde AI1
	rScaleAI1max 	: REAL :=50; //Max-värde AI1
	rScaleAI2min	: REAL :=0; //Min-värde AI1
	rScaleAI2max	: REAL :=2000; //Max-värde AI2
	tTimeout 		: TIME := T#5S; //Aktuell timeout
END_VAR
VAR_OUTPUT
	rAI1 			: REAL :=0; //Värde 0-100% för skrivning till AO1
	rAI2 			: REAL :=0; //Värde 0-100% för skrivning till AO2
	PV8 AT %M* 		: STRING := ' ';//Modbus konfiguering~wp:
	FAULT AT %M*  	: BOOL :=FALSE; //Kommunikationsfel Siox~wp:[trendoptions]i:300
END_VAR
VAR
	sIP 			: STRING(255) := ' ';
	sPort			: STRING(255) := ' ';
	sModbusID		: STRING(255) := ' ';
	sModbusLoop		: STRING(255) := ' ';
	sTemp 			: STRING(255) := ' ';
		
	bSekvensFlagga 	: BOOL :=FALSE;
	iStep			: INT :=0;
	bError			: BOOL := FALSE;
	bBusy			: BOOL := FALSE;
	
	fbKommTof		: Tof;
	fbKommTon 		: Ton;

	fbReadInputRegAI1_2 			: FB_MBReadInputRegs;
	fbReadWriteHoldingRegReal_AO1	: fbReadWriteHoldingRegReal;
	fbReadWriteHoldingRegReal_AO2	: fbReadWriteHoldingRegReal;
	nUnitIDinternal 				: UINT := 1;
	//Läs/skriv
	rWriteAO1						: REAL := 0;
	rWriteAO2						: REAL := 0;
	wArray1							: ARRAY[1..2] OF WORD;
	R_TRIG_Sekvens: R_TRIG;
	//Skalningar utgångar/ingångar
	FB_BA_Chrct02_A01 				: TC3_BA.FB_BA_Chrct02;
	FB_BA_Chrct02_A02 				: TC3_BA.FB_BA_Chrct02;
	FB_BA_Chrct02_AI1 				: TC3_BA.FB_BA_Chrct02;
	FB_BA_Chrct02_AI2 				: TC3_BA.FB_BA_Chrct02;
	rTemp1: REAL;
	rTemp2: REAL;
END_VAR

//Modbus konfiguering
	sIP := CONCAT (modbusTCP.sIPAddr, '');
	sPort := CONCAT ('<br>Port: ', UINT_TO_STRING(modbusTCP.nTCPPort));
	sModbusID := CONCAT('<br>Modbus-ID/SIOX-adr: ', UINT_TO_STRING(nUnitID));
	sModbusLoop := CONCAT('<br>Loop: ', INT_TO_STRING(modbusTCP.iModbusLoop));

	sTemp := sIP;
	sTemp := CONCAT(sTemp, sPort);
	sTemp := CONCAT(sTemp, sModbusID);
	sTemp := CONCAT(sTemp, sModbusLoop);
	
	PV8 := sTemp;

//Se till att det är ett giltligt modbus id
	nUnitIDinternal := INT_TO_UINT(LIMIT(1,nUnitID,256));
	
//Sekvens	
	bSekvensFlagga := oaksGVL.aBModbusSekvens[modbusTCP.iModbusLoop]= nUnitID;

	R_TRIG_Sekvens(CLK:= bSekvensFlagga, Q=>);

	CASE iStep OF

	0: 	//Start/reset
		bBusy := FALSE;
		IF bEnable AND R_TRIG_Sekvens.Q THEN
			iStep := 1;
			bError := FALSE;
			bBusy := TRUE;
		END_IF
	
	1: 	//Läs/skriv AO1
				 
		//Skalning AO1
		FB_BA_Chrct02_A01(
			rX:= rSetpointAO1, 
			rX01:= 0, 
			rX02:= 100, 
			rY01:= 0, 
			rY02:= 4096, 
			bLmt:= TRUE, 
			rY=> rWriteAO1, 
			bErr=> , 
			sErrDescr=> );
			
		fbReadWriteHoldingRegReal_AO1.bEnable := TRUE;
		
		//Skriv till AO1
		fbReadWriteHoldingRegReal_AO1(
			sIPAddr:= modbusTCP.sIPAddr, 
			nTCPPort:= modbusTCP.nTCPPort, 
			nUnitID:= nUnitIDinternal, 
			mBusAdr:= 12, 
			bEnable:= , // 
			tTimeout:= tTimeout, 
			rReal:= rWriteAO1, 
			uiFaktor:= 1, 
			bError=> , 
			bBusy=> , 
			bSuccess=> );
			
		//Error 
		IF fbReadWriteHoldingRegReal_AO1.bError THEN
			fbReadWriteHoldingRegReal_AO1(bEnable := FALSE);
			iStep := 99;
		END_IF
	
		//Gå till nästa steg
		IF NOT fbReadWriteHoldingRegReal_AO1.bBusy AND NOT fbReadWriteHoldingRegReal_AO1.bError THEN
			fbReadWriteHoldingRegReal_AO1(bEnable := FALSE);
			bError := FALSE;
			iStep := 2;
		END_IF;

	2: 	//Läs/skriv AO2 
		//Skalning AO2
		FB_BA_Chrct02_A02(
			rX:= rSetpointAO2, 
			rX01:= 0, 
			rX02:= 100, 
			rY01:= 0, 
			rY02:= 4096, 
			bLmt:= TRUE, 
			rY=> rWriteAO2, 
			bErr=> , 
			sErrDescr=> );
		
		fbReadWriteHoldingRegReal_AO2.bEnable := TRUE;	
			
		fbReadWriteHoldingRegReal_AO2(
			sIPAddr:= modbusTCP.sIPAddr, 
			nTCPPort:= modbusTCP.nTCPPort, 
			nUnitID:= nUnitIDinternal, 
			mBusAdr:= 13, 
			bEnable:= , 
			tTimeout:= tTimeout, 
			rReal:= rWriteAO2, 
			uiFaktor:= 1, 
			bError=> , 
			bBusy=> , 
			bSuccess=> );
		
		//Error 
		IF fbReadWriteHoldingRegReal_AO2.bError THEN
			fbReadWriteHoldingRegReal_AO2(bEnable := FALSE);
			iStep := 99;
		END_IF
	
		//Gå till nästa steg
		IF NOT fbReadWriteHoldingRegReal_AO2.bBusy AND NOT fbReadWriteHoldingRegReal_AO2.bError THEN
			fbReadWriteHoldingRegReal_AO2(bEnable := FALSE);
			bError := FALSE;
			iStep := 3;
		END_IF;

	3:	//Läsning AI1-2
	
		fbReadInputRegAI1_2.bExecute := TRUE;	
	
		fbReadInputRegAI1_2(
			sIPAddr:= modbusTCP.sIPAddr, 
			nTCPPort:= modbusTCP.nTCPPort, 
			nUnitID:= UINT_TO_BYTE(nUnitIDinternal), 
			nQuantity:=2 , 
			nMBAddr:=56, 
			cbLength:= SIZEOF(wArray1), 
			pDestAddr:= ADR(wArray1), 
			bExecute:= , 
			tTimeout:= T#3S, 
			bBusy=> , 
			bError=> , 
			nErrId=> , 
			cbRead=> );
								
		rTemp1 := fSignedConverter(WORD_TO_REAL(wArray1[1]));
		rTemp2 := fSignedConverter(WORD_TO_REAL(wArray1[2]));
			
		//Skalning AI1
		FB_BA_Chrct02_AI1( rX:= rTemp1, rX01:= 0, rX02:= 4096, rY01:= rScaleAI1min, rY02:= rScaleAI1max, bLmt:= TRUE, rY=> rAI1, bErr=> , sErrDescr=> );
		
		//Skalning AI2	
		FB_BA_Chrct02_AI2(rX:= rTemp2, rX01:= 0, rX02:= 4096, rY01:= rScaleAI2min, rY02:= rScaleAI2max, bLmt:= TRUE, rY=> rAI2, bErr=> , sErrDescr=> );

		//Error 
		IF fbReadInputRegAI1_2.bError THEN
			fbReadInputRegAI1_2(bExecute := FALSE);
			iStep := 99;
		END_IF
	
		//Gå till nästa steg
		IF NOT fbReadInputRegAI1_2.bBusy AND NOT fbReadInputRegAI1_2.bError THEN
			fbReadInputRegAI1_2(bExecute := FALSE);
			bError := FALSE;
			iStep := 20;
		END_IF;
		
	20: //Done
		bBusy := FALSE;
		iStep := 0;
		

	99: //Error handling
		bBusy := FALSE;
		bError := TRUE;
		iStep := 0;
		
END_CASE;
				
//Kommunikationsfel
	fbKommTof(IN:= bError, PT:=T#20S , Q=> , ET=> );
	fbKommTon(IN:=fbKommTof.Q , PT:=T#20M , Q=> , ET=> );
	FAULT :=fbKommTon.Q;
		
//Skriv upptagen till modbus-kö	
	oaksgvl.aBModbusBusyFlagga[modbusTCP.iModbusLoop,nUnitID] := bBusy;

END_FUNCTION_BLOCK

// oaksModbusLibrary/Siox/Via SX-Access/fbSioxDamperDUO
//OAKS AB 
//2020-06-10
//Funktionsblock för kommunikation med SIOX-DUO spjällmodul (2st spjäll).
FUNCTION_BLOCK fbSioxDamperDUO EXTENDS fbSioxDamperUNO

VAR_INPUT
	nSetpointDamper2Enable : BOOL; // Aktivera skrivning av 0-10V signal
	rSetpointDamper2 : REAL; // Värde 0-10V signal (0-100 skalning)
	nUnitIDDamper2 : UINT; // Modbus-id för spjäll vid 0-10V skrivning
END_VAR
VAR_OUTPUT
	DAMPER2_AL  AT %M*  : BOOL; //Driftfel spjäll 2~wp:
	DAMPER2_V0  AT %M*  : BOOL; //Stängtindikering spjäll 2~wp:[trendoptions]i:14400, t:1
	DAMPER2_V1  AT %M*  : BOOL; //Öppetindikering spjäll 2~wp:[trendoptions]i:14400, t:1
END_VAR
VAR

END_VAR

SUPER^();
//Modbus konfiguering
	DAMPER2_AL := wInternalWord.5;
	DAMPER2_V0 := wInternalWord.10;
	DAMPER2_V1 := wInternalWord.11;
	
	fbReadWriteHoldingRegDamper2.iWrite := REAL_TO_UINT(fScale2pInternalSetpoint(rX:=rSetpointDamper2 , Y1:=0 , Y2:=4096 , X1:=0 , X2:=100 ));

	fbReadWriteHoldingRegDamper2(
	sIPAddr:= sIPAddr, 
	nTCPPort:= nTCPPort, 
	nUnitID:= nUnitIDDamper2, 
	mBusAdr:=7 , 
	bEnable:= nSetpointDamper2Enable AND bSekvensFlagga, 
	iRead=> , 
	bError=> , 
	bBusy=> );

END_FUNCTION_BLOCK

// oaksModbusLibrary/Siox/Via SX-Access/fbSioxDamperUNO
//OAKS AB
//2022-03-17
//Funktionsblock för kommunikation med SIOX-UNO spjällmodul (1st spläll).
//Modbusloop är flyttad till fast 16 för att möjliggöra sekvens via adress istället för ID. 
FUNCTION_BLOCK fbSioxDamperUNO

VAR_INPUT
	


	sIPAddr : STRING := '192.168.1.32'; 
	nTCPPort : UINT := 502;
	nUnitID : BYTE := 60;
	iAdress : WORD := 257; //Startregister läsning
	nSetpointDamper1Enable : BOOL; // Aktivera skrivning av 0-10V signal
	rSetpointDamper1 : REAL;// Värde 0-10V signal (0-100 skalning)
	nUnitIDDamper1 : UINT; // Modbus-id för spjäll vid 0-10V skrivning
END_VAR
VAR_OUTPUT
	V AT %M*  : BOOL; //Standby bit (1=Standby)~wp:[trendoptions]i:14400, t:1
	PV5 AT %M*  : BOOL; //Motionskörning~wp:[trendoptions]i:14400, t:1
	AL AT %M*  : BOOL; //Övertemperatur (NTC)~wp:
	FAULT AT %M*  : BOOL; //Kommunikationsfel Siox~wp:
	GX_V  AT %M*  : BOOL; //Rökdetektor I drift~wp:[trendoptions]i:14400, t:1
	GX_AL  AT %M*  : BOOL; //Utlöst rökdetektor~wp:
	GX_AL1  AT %M*  : BOOL;  //Servicelarm rökdetektor~wp:
	GX_AL2  AT %M*  : BOOL; //Slingfel~wp:
	PV7 AT %M* : STRING;//Modbus adressering~wp:
	PV8 AT %M* : STRING;//Modbus konfiguering~wp:
	DAMPER1_AL  AT %M*  : BOOL; //Driftfel spjäll 1~wp:  
	DAMPER1_V0  AT %M*  : BOOL; //Stängtindikering spjäll 1~wp:[trendoptions]i:14400, t:1
	DAMPER1_V1  AT %M*  : BOOL; //Öppetindikering spjäll 1~wp:[trendoptions]i:14400, t:1
END_VAR
VAR
	iModbusLoop : INT :=1; //Modbusslinga
	offset : WORD;
	rTemp : REAL;
	iTemp : UINT;
	bSekvensFlagga : BOOL;	

	wInternalWord : WORD;
	fbKommTof: Tof;
	fbKommTon: Ton;
	FB_MBReadRegs01: FB_MBReadRegs;
	fbtoggle1 : fbToggle;
	
	sIP: STRING(255);
	sPort: STRING(255);
	sModbusID: STRING(255);
	sModbusLoop: STRING(255);
	sTemp : STRING(255);
	sTemp1 : STRING(255);
	wTemp : WORD;
	fbReadWriteHoldingRegDamper1: fbReadWriteHoldingReg;
	fbReadWriteHoldingRegDamper2: fbReadWriteHoldingReg;
END_VAR

iModbusLoop := 16; //Fast slinga

//Sekvens	
	bSekvensFlagga := oaksGVL.aBModbusSekvens[iModbusLoop] = WORD_TO_INT(iAdress);
	
	fbReadWriteHoldingRegDamper1.iWrite := REAL_TO_UINT(fScale2pInternalSetpoint(rX:=rSetpointDamper1 , Y1:=0 , Y2:=4096 , X1:=0 , X2:=100 ));

	fbReadWriteHoldingRegDamper1(
	sIPAddr:= sIPAddr, 
	nTCPPort:= nTCPPort, 
	nUnitID:= nUnitIDDamper1, 
	mBusAdr:=6 , 
	bEnable:= nSetpointDamper1Enable AND bSekvensFlagga, 
	iRead=> , 
	bError=> , 
	bBusy=> );

//Modbus konfiguering
	sIP := CONCAT (SIPAddr, '');
	sPort := CONCAT ('<br>Port: ', UINT_TO_STRING(nTCPPort));
	sModbusID := CONCAT('<br>Modbus-ID: ', UINT_TO_STRING(nUnitID));
	sModbusLoop := CONCAT('<br>Loop: ', INT_TO_STRING(iModbusLoop));

	sTemp := sIP;
	sTemp := CONCAT(sTemp, sPort);
	sTemp := CONCAT(sTemp, sModbusID);
	sTemp := CONCAT(sTemp, sModbusLoop);
	
	PV8 := sTemp;
	
	wTemp := iAdress -256; 
	sTemp := CONCAT('<br>Modbus-adress: ', WORD_TO_STRING(iAdress));
	sTemp := CONCAT(sTemp,'<br> Siox-adress: '); 
	PV7 := CONCAT(sTemp, WORD_TO_STRING(wTemp)); 
FB_MBReadRegs01(
	sIPAddr:= sIPAddr, 
	nTCPPort:= nTCPPort, 
	nUnitID:= nUnitID, 
	nQuantity:= 1, 
	nMBAddr:= iAdress, 
	cbLength:= SIZEOF(wInternalWord), 
	pDestAddr:=ADR(wInternalWord) , 
	bExecute:=bSekvensFlagga , 
	tTimeout:=T#4S , 
	bBusy=> , 
	bError=> , 
	nErrId=> , 
	cbRead=> );
	
	V := wInternalWord.0;
	PV5 := wInternalWord.4;
	AL :=  wInternalWord.7;
	DAMPER1_AL := wInternalWord.3;
	DAMPER1_V0 := wInternalWord.8;
	DAMPER1_V1 := wInternalWord.9;
	(* Används i DUO
	DAMPER2_AL := wInternalWord.5;
	DAMPER2_V0 := wInternalWord.10;
	DAMPER2_V1 := wInternalWord.11;
	*)
	GX_AL := wInternalWord.13;
	GX_AL1 := wInternalWord.14;
	GX_AL2 := wInternalWord.15;
	GX_V := wInternalWord.12;
	
	//Communication error
	fbKommTof(IN:=FB_MBReadRegs01.bError , PT:=T#20S , Q=> , ET=> );
	fbKommTon(IN:=fbKommTof.Q , PT:=T#20M , Q=> , ET=> );
	FAULT :=fbKommTon.Q;
		
//Write busy	
	oaksgvl.aBModbusBusyFlaggaAdresser[iModbusLoop-15,iAdress] := FB_MBReadRegs01.bBusy OR fbReadWriteHoldingRegDamper1.bBusy OR fbReadWriteHoldingRegDamper2.bBusy;

END_FUNCTION_BLOCK

// oaksModbusLibrary/Siox/fbSioxSxAcess
//OAKS AB
//2020-06-10
//Funktionsblock för kommunikation med SIOX-SX:ACESS centralenhet.
FUNCTION_BLOCK fbSioxSxAcess
VAR_INPUT
	sIPAddr : STRING := '127.0.0.1'; 
	nTCPPort : UINT :=502;
	nUnitID : UINT :=1;
	iModbusLoop : INT :=1; //Modbusslinga
	bEnableCommand: BOOL := FALSE; //Aktivering skrivning från modbus till register 44
END_VAR
VAR_OUTPUT
		
	PV10 AT %M* : STRING;//Modbus konfiguering~wp:
	FAULT AT %M* : BOOL;//Kommunikationsfel~wp:
	
END_VAR
VAR
	offset : WORD;
	rTemp : REAL;
	iTemp : UINT;
	bSekvensFlagga : BOOL;
			
	FB_MBReadRegs_ArrHolding1: FB_MBReadRegs;
	ArrHolding1 : ARRAY [0..10] OF WORD; //Holding
	
	FB_MBReadRegs_ArrHolding2: FB_MBReadRegs;
	ArrHolding2 : ARRAY [0..1] OF WORD; //Holding
		
	//Kommunikationsfel
	fbKommTof : tof; 
	fbKommTon : ton;
	
	sIP: STRING(255);
	sPort: STRING(255);
	sModbusID: STRING(255);
	sModbusLoop: STRING(255);
	sTemp : STRING(255);
	//Aktivering skrivning till register 44 (kommandoregistret i UNO/DUO). 
	fbReadWriteHoldingRegManover: fbReadWriteHoldingRegReal;
	rManover: REAL := 0;
END_VAR

VAR_OUTPUT
	
	V AT %M* : BOOL; //Driftindkering (DO4)~wp:[trendoptions]i:14400, t:1
	V3 AT %M* : BOOL; //DI1~wp:[trendoptions]i:14400, t:1
	V4 AT %M* : BOOL; //DI2~wp:[trendoptions]i:14400, t:1
	V5 AT %M* : BOOL; //DI3~wp:[trendoptions]i:14400, t:1
	V6 AT %M* : BOOL; //DI4~wp:	[trendoptions]i:14400, t:1
	PV1 AT %M* : REAL;//Antal brandlarm~wp:
	PV2 AT %M* : REAL;//Antal komm.fel moduler~wp:
	PV3 AT %M* : REAL;//Antal spjällfel~wp:
	PV4 AT %M* : REAL;//Antal servicelarm rökdetektorer~wp:
	PV5 AT %M* : REAL;//Antal moduler i motionsdrift~wp:
	AL AT %M* : BOOL; //Summalarm (DO1)~wp:
	AL1 AT %M* : BOOL; //Brandlarm (DO2)~wp:
	AL2 AT %M* : BOOL; //Servicelarm (DO3)~wp:

END_VAR

//General
	offset := 0;
//Sekvens	
	bSekvensFlagga := oaksGVL.aBModbusSekvens[iModbusLoop] = UINT_TO_INT(nUnitID);
//Modbus konfiguering
	sIP := CONCAT (SIPAddr, '');
	sPort := CONCAT (' <br>Port: ', UINT_TO_STRING(nTCPPort)); 								
	sModbusID := CONCAT(' <br>ID: ', UINT_TO_STRING(nUnitID));
	sModbusLoop := CONCAT(' <br>Loop: ', INT_TO_STRING(iModbusLoop));	

	sTemp := sIP;
	sTemp := CONCAT(sTemp, sPort);
	sTemp := CONCAT(sTemp, sModbusID);
	sTemp := CONCAT(sTemp, sModbusLoop);
	
	PV10 := sTemp;
	
///////////////
//WRITE
//////////////

IF bEnableCommand THEN
	rManover := 1;
ELSE
	rManover := 0;
END_IF

	//Skriv
	fbReadWriteHoldingRegManover(
	sIPAddr:= sIPAddr, 
	nTCPPort:= nTCPPort, 
	nUnitID:= nUnitID, 
	mBusAdr:=63 , 
	bEnable:= bSekvensFlagga,
	tTimeout:= T#5S, 
	rReal:= rManover, 
	uiFaktor:= 1, 
	bError=> , 
	bBusy=> ); 	

///////////////		
//READ
///////////////		
	
	//Read Holding 0-10
	FB_MBReadRegs_ArrHolding1(
	sIPAddr:= sIpAddr, 
	nTCPPort:= INT_TO_UINT(nTCPPort), 
	nUnitID:= INT_TO_BYTE(nUnitID), 
	nQuantity:= 5, 
	nMBAddr:= 80 + offset, 
	cbLength:= SIZEOF(ArrHolding1), 
	pDestAddr:= ADR(ArrHolding1), 
	bExecute:= bSekvensFlagga, 
	tTimeout:= T#3S, 
	bBusy=> , 
	bError=> , 
	nErrId=> , 
	cbRead=> );
	
		//Values
		PV1 := ArrHolding1[0]; //0
		PV2 := ArrHolding1[1]; //1
		PV3 := ArrHolding1[2]; //2
		PV4 := ArrHolding1[3]; //3
		PV5 := ArrHolding1[4]; //4
		//ArrHolding1[5]; //5
		//ArrHolding1[6]; //6
		//ArrHolding1[7]; //7
		//ArrHolding1[8]; //8
		//ArrHolding1[8]; //9
		//ArrHolding1[8]; //10

	//Read Holding 0-10
	FB_MBReadRegs_ArrHolding2(
	sIPAddr:= sIpAddr, 
	nTCPPort:= INT_TO_UINT(nTCPPort), 
	nUnitID:= INT_TO_BYTE(nUnitID), 
	nQuantity:= 2, 
	nMBAddr:= 56 + offset, 
	cbLength:= SIZEOF(ArrHolding2), 
	pDestAddr:= ADR(ArrHolding2), 
	bExecute:= bSekvensFlagga, 
	tTimeout:= T#3S, 
	bBusy=> , 
	bError=> , 
	nErrId=> , 
	cbRead=> );
		
	//Values
	AL := ArrHolding2[0].0; //0
	AL1 := ArrHolding2[0].1; //1
	AL2 := ArrHolding2[0].2; //2
	V := ArrHolding2[0].3; //3
	// := ArrHolding2[0].4; //4
	// := ArrHolding2[0].5; //5
	// := ArrHolding2[0].6; //6
	
	V3 := ArrHolding2[1].0; //0
	V4 := ArrHolding2[1].1; //1
	V5 := ArrHolding2[1].2; //2
	V6 := ArrHolding2[1].3; //3
			
//Communication error
	fbKommTof(IN:=FB_MBReadRegs_ArrHolding1.bError OR FB_MBReadRegs_ArrHolding2.bError, PT:=T#20S , Q=> , ET=> );
	fbKommTon(IN:=fbKommTof.Q , PT:=T#20M , Q=> , ET=> );
	FAULT :=fbKommTon.Q;
		
//Write busy	
	oaksgvl.aBModbusBusyFlagga[iModbusLoop,nUnitID] := FB_MBReadRegs_Arrholding1.bBusy OR FB_MBReadRegs_Arrholding2.bBusy;

END_FUNCTION_BLOCK

// oaksModbusLibrary/Swegon/fbSwegonGoldCdOperationLevel
// Skrivning till Swegon Gold C/D driftval.
// Välj för respektive läge vilken hastighet som skall skickas. 
//Communication operation mode 
//Setting of unit operation mode from communication. 
//0=Auto operation (Normal stop when time channels are deactivated). 
//1=Communication stop 1. 
//2=Communication Iow speed. , 3=Communication high speed. 
//4=Communication stop 2 (New in PV 5.00). Intermittent night heat and mornin boost functions works at stop 2. 
FUNCTION_BLOCK fbSwegonGoldCdOperationLevel
VAR_INPUT
	sIPAddr : STRING; // Ip-adress till gold-aggregat
	usiTimechannel : USINT := 3; // Välj hastighet vid tidkanal 2=Communication Iow speed. , 3=Communication high speed. 
	bTimechannel : BOOL; // Ingång för knytning av tidkanal
	usiPushbutton : USINT := 3; // Välj hastighet vid tryckknappsdrift.  2=Communication Iow speed. , 3=Communication high speed. 
	bPushbutton : BOOL; // Ingång för knytning av tryckkanpp för förlängd drift
	usiPrescence : USINT := 2; // Välj hastighet vid närvarodrift 2=Communication Iow speed. , 3=Communication high speed. 
	bPrescence : BOOL; // Ingång för knytning av närvarosensor eller valfritt. Bara att lämna den tom om den ej används.
	usiStopMode : USINT := 1; // Välj stoppläge  1=Communication stop 1. , 4=Communication stop 2 (New in PV 5.00). Intermittent night heat and mornin boost functions works at stop 2. 
END_VAR
VAR_OUTPUT
	PV8 : STRING; //Modbus konfiguering~wp:
	FAULT AT %M* : BOOL;//Kommunikationsfel Swegon Gold Ventilationsaggregat~wp:
END_VAR
VAR
	//Kommunikationsfel
	fbKommTof : tof; 
	fbAlarmCommunicationError : fbAlarm;
	fbToggle_run: fbToggle;
	fbReadWriteHoldingSwegonGoldHoldingRegAdr174 : fbReadWriteHoldingReg;
END_VAR
VAR PERSISTENT
	tToggleTid : TIME := T#3S;
END_VAR
VAR // added by the converter: edge detectors and wires of the graphical bodies
    _w1, _w3 : ANY;
    _w2 : BOOL;
END_VAR

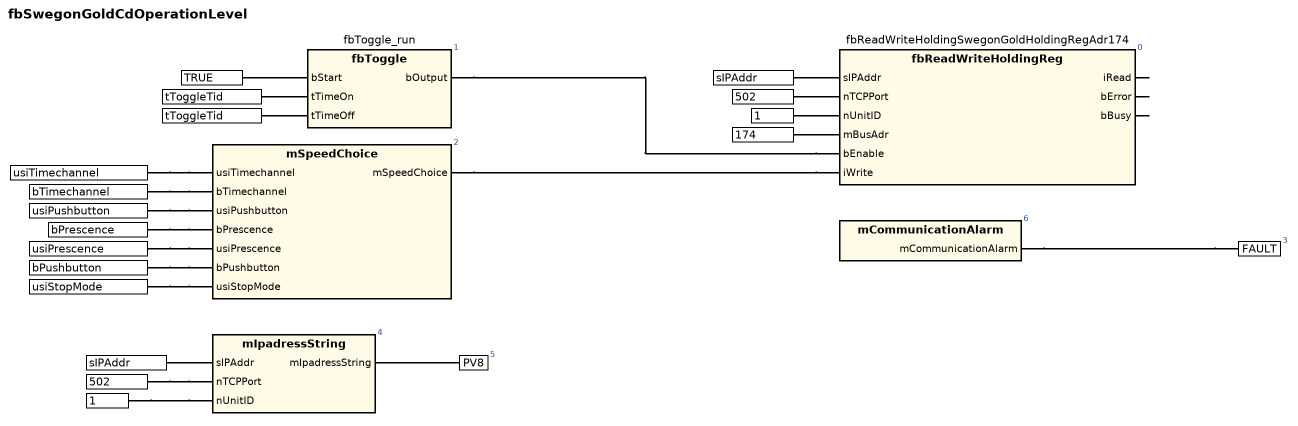
// note: 13 stored wires end on pins the file does not list and are not shown
fbReadWriteHoldingSwegonGoldHoldingRegAdr174(
    sIPAddr := sIPAddr,
    nTCPPort := 502,
    nUnitID := 1,
    mBusAdr := 174,
    bEnable := fbToggle_run.bOutput,
    iWrite := _w1); // fbReadWriteHoldingReg
fbToggle_run(bStart := TRUE, tTimeOn := tToggleTid, tTimeOff := tToggleTid); // fbToggle
_w1 := mSpeedChoice(usiTimechannel := usiTimechannel, bTimechannel := bTimechannel, usiPushbutton := usiPushbutton, bPrescence := bPrescence, usiPrescence := usiPrescence, bPushbutton := bPushbutton, usiStopMode := usiStopMode);
FAULT := _w2;
_w3 := mIpadressString(sIPAddr := sIPAddr, nTCPPort := 502, nUnitID := 1);
PV8 := _w3;
_w2 := mCommunicationAlarm();

METHOD mCommunicationAlarm : BOOL
VAR 

END_VAR
	//Communication error
	fbKommTof(IN:=fbReadWriteHoldingSwegonGoldHoldingRegAdr174.bError , PT:=T#20S , Q=> , ET=> );
	fbAlarmCommunicationError(bInput:=fbKommTof.Q , tAlarmDelay:=T#60S , bAutoReset:=TRUE , bAlarmOutput=> );
	mCommunicationAlarm :=fbAlarmCommunicationError.bAlarmOutput;
END_METHOD

METHOD mIpadressString : STRING
VAR_INPUT
	sIPAddr : STRING := ''; 
	nTCPPort : UINT;
	nUnitID : UINT :=1;
END_VAR
VAR
	sIP: STRING(255);
	sPort: STRING(255);
	sModbusID: STRING(255);
	sTemp : STRING(255);
END_VAR
//Modbus konfiguering
	sIP := CONCAT (SIPAddr, '');
	sPort := CONCAT ('<br>Port: ', UINT_TO_STRING(nTCPPort)); 								
	sModbusID := CONCAT('<br>ID: ', UINT_TO_STRING(nUnitID));

	sTemp := sIP;
	sTemp := CONCAT(sTemp, sPort);
	sTemp := CONCAT(sTemp, sModbusID);
	
	mIpadressString := sTemp;
END_METHOD

METHOD PRIVATE mSpeedChoice : USINT
VAR_INPUT
	usiTimechannel : USINT;
	bTimechannel : BOOL;
	usiPushbutton : USINT;
	bPushbutton : BOOL;
	usiPrescence : USINT;
	bPrescence : BOOL;
	usiStopMode : USINT;
END_VAR
IF bTimechannel THEN
	mSpeedChoice := usiTimechannel;
ELSIF bPushbutton THEN
	mSpeedChoice := usiPushbutton;	
ELSIF bPrescence THEN
	mSpeedChoice := usiPrescence;	
ELSE 
	mSpeedChoice := usiStopMode;
END_IF
END_METHOD

END_FUNCTION_BLOCK

// oaksModbusLibrary/Swegon/fbSwegonGoldIndication
FUNCTION_BLOCK fbSwegonGoldIndication
VAR_INPUT
	sIPAddr : STRING := ''; 
	nTCPPort : UINT := 502;
	nUnitID : UINT :=1;
	tTimeOut : TIME := T#20M;	
	tToggleTime : TIME := T#1s;
END_VAR
VAR_OUTPUT
		
	PV8 AT %M* : STRING;//Modbus konfiguering~wp:
	FAULT AT %M* : BOOL;//Kommunikationsfel~wp:
	
	HEAT_CIRCPUMP_V AT %M* : BOOL;//Driftindikering pump värmebatteri~wp:[trendoptions]i:14400, t:1

	SUPPLY_FAN_V AT %M* : BOOL;//Driftindikering tilluftsfläkt~wp:[trendoptions]i:14400, t:1
	SUPPLY_FAN_OP AT %M* : REAL;//Utsignal tilluftsfläkt~wp:[trendoptions]i:300	[unit]%[format]0
	EXHAUST_FAN_V AT %M* : BOOL;//Driftindikering frånluftsfläkt~wp:[trendoptions]i:14400, t:1
	EXHAUST_FAN_OP AT %M* : REAL;//Utsignal tilluftsfläkt~wp:[trendoptions]i:300[unit]%[format]0
	
	HEAT_OP AT %M* : REAL;//Utsignal värme~wp:[trendoptions]i:300[unit]%[format]0
	
	COOL_OP AT %M* : REAL;//Utsignal kyla~wp:[trendoptions]i:300[unit]%[format]0
END_VAR
VAR
	rTemp : REAL;
	wSupfan : WORD;
	wExhfan : WORD;	

	fbToggle01 :	fbToggle;

	FB_MBReadCoilsHeatpump : FB_MBReadCoils;
	
	offset : WORD;
	iTemp : UINT;

		
	//Kommunikationsfel
	fbKommTof : tof; 
	fbKommTon : fbAlarm;
	
	sIP: STRING(255);
	sPort: STRING(255);
	sModbusID: STRING(255);
	sModbusLoop: STRING(255);
	sTemp : STRING(255);
	
	
	FB_MBReadInputRegsSupplyFan: FB_MBReadInputRegs;
	FB_MBReadInputRegsExhFan: FB_MBReadInputRegs;
	
	FB_MBReadInputRegsCoolOutput: FB_MBReadInputRegs;
	wCoolOutput : WORD;

	FB_MBReadInputRegsHeatOutput: FB_MBReadInputRegs;
	wHeatOutput : WORD;	
END_VAR

//General
	offset := 0;
//Modbus konfiguering
	sIP := CONCAT (SIPAddr, '');
	sPort := CONCAT ('<br>Port: ', UINT_TO_STRING(nTCPPort)); 								
	sModbusID := CONCAT('<br>ID: ', UINT_TO_STRING(nUnitID));

	sTemp := sIP;
	sTemp := CONCAT(sTemp, sPort);
	sTemp := CONCAT(sTemp, sModbusID);
	
	PV8 := sTemp;
	fbToggle01(bStart:=TRUE , tTimeOn:=tToggleTime , tTimeOff:=tToggleTime , bOutput=> );

(*P1_V		10038	DIGITAL	0	1	0	1		0	Indikering Cirkpump Värme*)
	FB_MBReadCoilsHeatpump(
	sIPAddr:= sIpAddr, 
	nTCPPort:= INT_TO_UINT(nTCPPort), 
	nUnitID:= INT_TO_BYTE(nUnitID), 
	nQuantity:= 1, 
	nMBAddr:= 37, 
	cbLength:=SIZEOF(HEAT_CIRCPUMP_V) , 
	pDestAddr:=ADR(HEAT_CIRCPUMP_V) , 
	bExecute:= fbToggle01.bOutput, 
	tTimeout:= T#3S, 
	bBusy=> , 
	bError=> , 
	nErrId=> , 
	cbRead=> );
//TF1_OP		30037	INT	0	10000	0	100	%	0	Utsignal Tilluftsfläkt
	FB_MBReadInputRegsSupplyFan(
	sIPAddr:= sIpAddr, 
	nTCPPort:= INT_TO_UINT(nTCPPort), 
	nUnitID:= INT_TO_BYTE(nUnitID), 
	nQuantity:=1 , 
	nMBAddr:= 36, 
	cbLength:=SIZEOF(wSupfan), 
	pDestAddr:=ADR(wSupfan) ,
	bExecute:= fbToggle01.bOutput, 
	tTimeout:= T#3S, 
	bBusy=> , 
	bError=> , 
	nErrId=> , 
	cbRead=> );
	
	rTemp := 	WORD_TO_REAL(wSupfan);
	SUPPLY_FAN_OP := rTemp / 100;
	SUPPLY_FAN_V := wSupfan > 0;
//FF1_OP		30038	INT	0	10000	0	100	%	0	Utsignal Frånluftsfläkt
	FB_MBReadInputRegsExhFan(
	sIPAddr:= sIpAddr, 
	nTCPPort:= INT_TO_UINT(nTCPPort), 
	nUnitID:= INT_TO_BYTE(nUnitID), 
	nQuantity:=1 , 
	nMBAddr:= 37, 
	cbLength:=SIZEOF(wExhfan), 
	pDestAddr:=ADR(wExhfan) ,
	bExecute:= fbToggle01.bOutput, 
	tTimeout:= T#3S, 
	bBusy=> , 
	bError=> , 
	nErrId=> , 
	cbRead=> );
	
	rTemp := 	WORD_TO_REAL(wExhfan);
	EXHAUST_FAN_OP := rTemp / 100;
	EXHAUST_FAN_V := wSupfan > 0;

// COOL_OP		30102	INT	0	10000	0	100	%	0	Utsignal Kyla
	FB_MBReadInputRegsCoolOutput(
	sIPAddr:= sIpAddr, 
	nTCPPort:= INT_TO_UINT(nTCPPort), 
	nUnitID:= INT_TO_BYTE(nUnitID), 
	nQuantity:=1 , 
	nMBAddr:= 101, 
	cbLength:=SIZEOF(wCoolOutput), 
	pDestAddr:=ADR(wCoolOutput) ,
	bExecute:= fbToggle01.bOutput, 
	tTimeout:= T#3S, 
	bBusy=> , 
	bError=> , 
	nErrId=> , 
	cbRead=> );
	rTemp := 	WORD_TO_REAL(wCoolOutput);
	COOL_OP := rTemp / 100;
// HEAT_OP		30094	INT	0	10000	0	100	%	0	Utsignal Värme	
	FB_MBReadInputRegsHeatOutput(
	sIPAddr:= sIpAddr, 
	nTCPPort:= INT_TO_UINT(nTCPPort), 
	nUnitID:= INT_TO_BYTE(nUnitID), 
	nQuantity:=1 , 
	nMBAddr:= 93, 
	cbLength:=SIZEOF(wHeatOutput), 
	pDestAddr:=ADR(wHeatOutput) ,
	bExecute:= fbToggle01.bOutput, 
	tTimeout:= T#3S, 
	bBusy=> , 
	bError=> , 
	nErrId=> , 
	cbRead=> );
	rTemp := 	WORD_TO_REAL(wHeatOutput);
	HEAT_OP := rTemp / 100;
//Communication error
	fbKommTof(IN:=FB_MBReadCoilsHeatpump.bError , PT:=T#20S , Q=> , ET=> );
	fbKommTon(bInput:=fbKommTof.Q , tAlarmDelay:=tTimeOut , bAutoReset:= , bAlarmOutput=> );
	FAULT :=fbKommTon.bAlarmOutput;

END_FUNCTION_BLOCK

// oaksModbusLibrary/Swegon/fbSwegonGoldOperationLevel
// Skrivning till Swegon Gold E/F driftval 0=auto, 1=total stop, 2=low speed, 3=high speed, 4=normal stop, 5=extended normal stop.
// Välj för respektive läge vilken hastighet som skall skickas. 
//There are five different operating modes:
//Total stop = The AHU is completely stopped, no internal automatic functions or external control commands can start the AHU.
//Normal Stop = The AHU has stopped, however all the internal and external automatic functions oversteer the stop.
//Extended Normal Stop = The AHU has stopped, however all the internal and external automatic functions, with exception of Summer night cool, oversteer the stop.
//Low speed = The AHU is running at the preset low speed setting.
//High speed = The AHU is running at the preset high speed setting.


FUNCTION_BLOCK fbSwegonGoldOperationLevel
VAR_INPUT
	sIPAddr : STRING; // Ip-adress till gold-aggregat
	usiTimechannel : USINT := 3; // Välj hastighet vid tidkanal 0=auto, 1=total stop, 2=low speed, 3=high speed, 4=normal stop, 5=extended normal stop.
	bTimechannel : BOOL; // Ingång för knytning av tidkanal
	usiPushbutton : USINT := 3; // Välj hastighet vid tryckknappsdrift 0=auto, 1=total stop, 2=low speed, 3=high speed, 4=normal stop, 5=extended normal stop.
	bPushbutton : BOOL; // Ingång för knytning av tryckkanpp för förlängd drift
	usiPrescence : USINT := 2; // Välj hastighet vid närvarodrift 0=auto, 1=total stop, 2=low speed, 3=high speed, 4=normal stop, 5=extended normal stop.
	bPrescence : BOOL; // Ingång för knytning av närvarosensor eller valfritt. Bara att lämna den tom om den ej används.
	usiStopMode : USINT := 4; // Välj stoppläge  1=total stop (ingen aggregatsstyrd nattkyla/nattanvärmning eller möjlighet till förlängd drift) 4=normal stop (med aggregatsstyrd nattkyla/nattanvärmning och möjlighet till förlängd drift), 5=extended normal stop (ingen aggregatsstyrd nattkyla/nattanvärmning MEN möjlighet till förlängd drift)
END_VAR
VAR_OUTPUT
	PV8 : STRING; //Modbus konfiguering~wp:
	FAULT AT %M* : BOOL;//Kommunikationsfel Swegon Gold Ventilationsaggregat~wp:
END_VAR
VAR
	//Kommunikationsfel
	fbKommTof : tof; 
	fbAlarmCommunicationError : fbAlarm;
	fbToggle_run: fbToggle;
	fbReadWriteHoldingSwegonGoldHoldingRegAdr792 : fbReadWriteHoldingReg;
END_VAR
VAR PERSISTENT
	tToggleTid : TIME := T#3S;
END_VAR
VAR // added by the converter: edge detectors and wires of the graphical bodies
    _w1, _w2, _w3 : ANY;
END_VAR

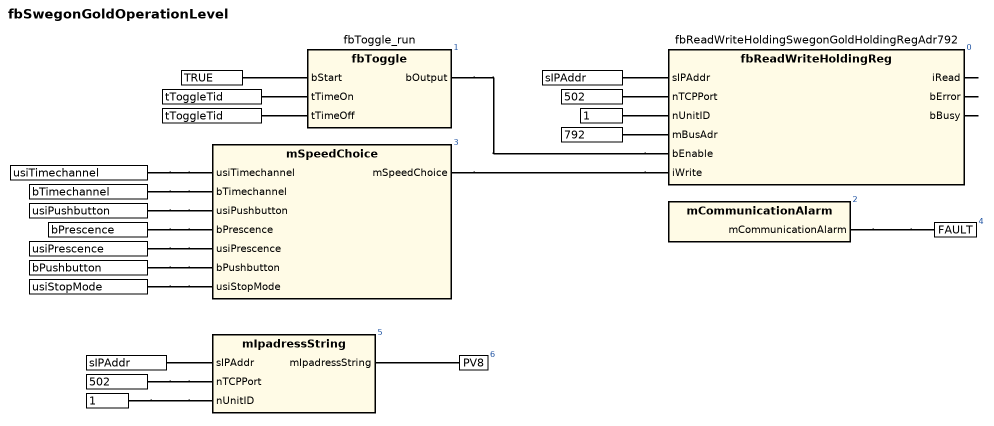
// note: 6 stored wires end on pins the file does not list and are not shown
fbReadWriteHoldingSwegonGoldHoldingRegAdr792(
    sIPAddr := sIPAddr,
    nTCPPort := 502,
    nUnitID := 1,
    mBusAdr := 792,
    bEnable := fbToggle_run.bOutput,
    iWrite := _w1); // fbReadWriteHoldingReg
fbToggle_run(bStart := TRUE, tTimeOn := tToggleTid, tTimeOff := tToggleTid); // fbToggle
_w2 := mCommunicationAlarm();
_w1 := mSpeedChoice(usiTimechannel := usiTimechannel, bTimechannel := bTimechannel, usiPushbutton := usiPushbutton, bPrescence := bPrescence, usiPrescence := usiPrescence, bPushbutton := bPushbutton, usiStopMode := usiStopMode);
FAULT := _w2;
_w3 := mIpadressString(sIPAddr := sIPAddr, nTCPPort := 502, nUnitID := 1);
PV8 := _w3;

METHOD mCommunicationAlarm : BOOL
VAR 

END_VAR
	//Communication error
	fbKommTof(IN:=fbReadWriteHoldingSwegonGoldHoldingRegAdr792.bError , PT:=T#20S , Q=> , ET=> );
	fbAlarmCommunicationError(bInput:=fbKommTof.Q , tAlarmDelay:=T#60S , bAutoReset:=TRUE , bAlarmOutput=> );
	mCommunicationAlarm :=fbAlarmCommunicationError.bAlarmOutput;
END_METHOD

METHOD mIpadressString : STRING
VAR_INPUT
	sIPAddr : STRING := ''; 
	nTCPPort : UINT;
	nUnitID : UINT :=1;
END_VAR
VAR
	sIP: STRING(255);
	sPort: STRING(255);
	sModbusID: STRING(255);
	sTemp : STRING(255);
END_VAR
//Modbus konfiguering
	sIP := CONCAT (SIPAddr, '');
	sPort := CONCAT ('<br>Port: ', UINT_TO_STRING(nTCPPort)); 								
	sModbusID := CONCAT('<br>ID: ', UINT_TO_STRING(nUnitID));

	sTemp := sIP;
	sTemp := CONCAT(sTemp, sPort);
	sTemp := CONCAT(sTemp, sModbusID);
	
	mIpadressString := sTemp;
END_METHOD

METHOD PRIVATE mSpeedChoice : USINT
VAR_INPUT
	usiTimechannel : USINT;
	bTimechannel : BOOL;
	usiPushbutton : USINT;
	bPushbutton : BOOL;
	usiPrescence : USINT;
	bPrescence : BOOL;
	usiStopMode : USINT;
END_VAR
IF bTimechannel THEN
	mSpeedChoice := usiTimechannel;
ELSIF bPushbutton THEN
	mSpeedChoice := usiPushbutton;	
ELSIF bPrescence THEN
	mSpeedChoice := usiPrescence;	
ELSE 
	mSpeedChoice := usiStopMode;
END_IF
END_METHOD

END_FUNCTION_BLOCK

// oaksModbusLibrary/Swegon/fbSwegonReact
FUNCTION_BLOCK fbSwegonReact
VAR_INPUT
	sIPAddr : STRING := ''; 
	nTCPPort : UINT;
	nUnitID : UINT;
	nModbusLoop : UINT := 1;
	rSetpoint : REAL; // Flödessignal mellan 0-100
	wOperationMode : WORD := 1; // Driftläge (0 = börvärde via analog in 0-10V, 1 = börvärde via modbus)
	wMode : WORD := 0; //Överstyrning spjälläge 0: None 1: Open 2: Close 3: Min 4: Max 5: Mid
	bMode : BOOL := FALSE; //Överstyrning spjälläge aktiverad
	SP1 AT %M*  : REAL; //Inställt min. flöde~wp:[unit]l/s[format]0
	SP2 AT %M*  : REAL; //Inställt max. flöde~wp:[unit]l/s[format]0

END_VAR
VAR_OUTPUT
	CSP AT %M*  : REAL; //Aktuellt börvärde~wp:[trendoption]i:300[unit]l/s[format]0
	OP AT %M*  : REAL; //Spjällposition relativ~wp:[trendoption]i:300[unit]%[format]0
	PV4 AT %M*  : REAL; //Uträknat börvärde~wp:[trendoption]i:300[unit]%[format]0
	AL8 AT %M*  : BOOL; //Handställningslarm~wp:
	PV AT %M*  : REAL; // Ärvärde flöde~wp:[trendoption]i:300[unit]l/s[format]0
	PV7 AT %M* : BOOL;//Senaste läsning OK~wp:
	PV8 AT %M* : STRING;//Modbus konfiguering~wp:
	FAULT AT %M* : BOOL;//Kommunikationsfel~wp:
END_VAR
VAR
	wOperationModeInternal : WORD; // Driftläge (0 = börvärde via analog in 0-10V, 1 = börvärde via modbus) intern hantering för handställning. Blir 1 oavsett läge ifall variabel M är TRUE

	bFlodesBalanseringAktiv : BOOL := FALSE; // Aktiveras då man kör metod mFlodesBalansering 
	rFlodesBalansering  : REAL;  // Detta börvärde används då man kör metod mFlodesBalansering 

